# B&R Automation Studio project 8238 (part 30)

#### SupertrackLiftingStaticBag.st
```iecst
(* TODO: Add your comment here *)
FUNCTION_BLOCK SupertrackLiftingStaticBag

	messages ACCESS p_messages;

	// Device State Machine
	IF reset THEN
		IF rail_mt THEN
			udp_data.state := state := ReadyToReceive;
		ELSE
			udp_data.state := state := Loaded;
		END_IF;
	END_IF;
	IF udp_data.state = 0 THEN udp_data.state := state := ReadyToReceive; END_IF;

	// Debounce ON
	DBNC_up_timer(IN := up_raw, PT := DBNC_up_time);
	up := DBNC_up_timer.Q;

	DBNC_down_timer(IN := down_raw, PT := DBNC_down_time);
	down := DBNC_down_timer.Q;

	CASE udp_data.state OF
		Closed:
			IF dischargerRailSlingReady AND input_enabled AND NOT(safety_zone) AND NOT(halted) THEN
				udp_data.state := state := PreparingToLift;
			END_IF;

		PreparingToLift:
			IF PreparingToLiftTimer.Q THEN udp_data.state := state := Lifting; END_IF;

		Lifting:
			IF up THEN udp_data.state := state := DoneLifting; END_IF;

		DoneLifting:
			IF DoneLiftingTimer.Q THEN udp_data.state := state := InReceivePosition; END_IF;

		InReceivePosition:
			IF input_enabled AND NOT(safety_zone) AND NOT(halted) THEN
				udp_data.state := state := ReadyToReceive;
			ELSIF NOT(input_enabled) THEN
				udp_data.state := state := PreparingToLower;
			END_IF;

		ReadyToReceive:
			IF man_send THEN
				udp_data.state := state := Receiving;
			ELSIF NOT(input_enabled) OR safety_zone OR halted THEN
				udp_data.state := state := InReceivePosition;
			END_IF;

		Receiving:
			IF ReceivingTimer.Q THEN udp_data.state := state := PreparingToLower; END_IF;

		PreparingToLower:
			IF PreparingToLowerTimer.Q THEN udp_data.state := state := Lowering; END_IF;

		Lowering:
			IF down THEN udp_data.state := state := DoneLowering; END_IF;

		DoneLowering:
			IF DoneLoweringTimer.Q THEN
				IF rail_mt THEN
					udp_data.state := state := Closed;
				ELSE
					udp_data.state := state := Loaded;
				END_IF;
			END_IF;

		Loaded:
			IF NOT(halted) AND NOT(safety_zone) AND NOT(stopped) THEN
				udp_data.state := state := ReadyToTransfer;
			END_IF;

		ReadyToTransfer:
			IF open_signal OR man_open OR open_pendant THEN
				delete_latch := TRUE;
				udp_data.state := state := Unclamping;
			ELSIF halted OR stopped OR safety_zone THEN
				udp_data.state := state := Loaded;
			END_IF;

		Unclamping:
			IF UnclampingTimer.Q THEN udp_data.state := state := Opening; END_IF;

		Opening:
			IF static_open THEN udp_data.state := state := Transferring; END_IF;

		Transferring:
			IF man_send THEN udp_data.state := state := Closing; END_IF;

		Closing:
			IF static_close THEN udp_data.state := state := Closed; END_IF;

	END_CASE;

	clamp := udp_data.state = Unclamping OR udp_data.state = Opening OR udp_data.state = Transferring OR udp_data.state = Closing;
	open := udp_data.state = Opening;
	close := udp_data.state = Closing;

	lift_clamp := (
	udp_data.state = PreparingToLift
	OR udp_data.state = Lifting
	OR udp_data.state = PreparingToLower
	OR udp_data.state = Lowering
	);

	fire_up := (
	udp_data.state = Lifting
	OR udp_data.state = InReceivePosition
	OR udp_data.state = ReadyToReceive
	OR udp_data.state = Receiving
	OR udp_data.state = PreparingToLower
	);

	fire_down := NOT(fire_up);

	// Control Timers
	ReceivingTimer(IN := (udp_data.state = Receiving), PT := ReceivingTime);
	PreparingToLiftTimer(IN := (udp_data.state = PreparingToLift), PT := PreparingToLiftTime);
	PreparingToLowerTimer(IN := (udp_data.state = PreparingToLower), PT := PreparingToLowerTime);
	UnclampingTimer(IN := (udp_data.state = Unclamping), PT := UnclampingTime);
	DoneLiftingTimer(IN := udp_data.state = DoneLifting, PT := DoneLiftingTime);
	DoneLoweringTimer(IN := udp_data.state = DoneLowering, PT := DoneLoweringTime);

	// Comm Logic
	bring_ok := udp_data.state = Closing OR udp_data.state = Closed;
	waiting := FALSE;
	man_open := man_send := FALSE;
	sling_ready := udp_data.state = ReadyToTransfer;
	dischargerRailReceiveSignal := udp_data.state = DoneLowering;

	IF rail_mt THEN delete_latch := FALSE; END_IF;

	udp_data.alarm := alarm := FALSE;
	udp_data.warning_com.0 := warning_com.0 := FALSE;
	udp_data.warning_com.1 := warning_com.1 := FALSE;
	udp_data.warning_com.12 := warning_com.12 := delete_latch;
	udp_data.warning_com.14 := warning_com.14 := sling_ready;

	//messages.Write := 0;
	//IF UnexpectedBagTimer.Q   THEN messages.Write := BIT_SET(messages.Write,UNEXPECTED_BAG); END_IF;
	//IF MissingBagTimer.Q      THEN messages.Write := BIT_SET(messages.Write,MISSING_BAG); END_IF;

	// Always clear acknowledgements
	//brsmemset(ADR(messages.Read[0]),0,SIZEOF(messages.Read));

END_FUNCTION_BLOCK
```

#### SupertrackBinTransfer.st
```iecst
(* TODO: Add your comment here *)
FUNCTION_BLOCK SupertrackBinTransfer

	messages ACCESS p_messages;

	// Debounce Inputs
	DBNC_front_timer(IN := front_raw, PT := DBNC_front_time);
	front := DBNC_front_timer.Q;

	DBNC_arrive_timer(IN := arrive_raw, PT := DBNC_arrive_time);
	arrive := DBNC_arrive_timer.Q;

	DBNC_after_timer(IN := after_raw, PT := DBNC_after_time);
	after := DBNC_after_timer.Q;

	DBNC_mid_timer(IN := mid_raw, PT := DBNC_mid_time);
	mid_sensor := DBNC_mid_timer.Q;

	// Device State Machine
	IF reset THEN
		IF rail_mt AND NOT(going_to) THEN
			udp_data.state := state := ReadyToReceive;
		ELSIF NOT(rail_mt) THEN
			udp_data.state := state := ReadyToLoad;
		END_IF;
	END_IF;
	IF udp_data.state = 0 THEN udp_data.state := state := ReadyToReceive; END_IF;

	CASE udp_data.state OF
		ReadyToReceive:
			IF going_to THEN
				udp_data.state := state := Receiving;
			ELSIF NOT(rail_mt) THEN
				udp_data.state := state := ReadyToLoad;
			END_IF;

		Receiving:
			IF mid_sensor THEN
				udp_data.state := state := CatchRear;
			ELSIF NOT(going_to) THEN
				udp_data.state := state := ReadyToReceive;
			END_IF;

		CatchRear:
			IF NOT(rail_mt) THEN
				udp_data.state := state := ReadyToLoad;
			ELSIF NOT(going_to) THEN
				udp_data.state := state := ReadyToReceive;
			END_IF;

		ReadyToLoad:
			IF onoff AND NOT(halted) THEN
				udp_data.state := state := Stabilizing;
			ELSIF rail_mt AND NOT(front) THEN
				udp_data.state := state := ReadyToReceive;
			END_IF;

		Stabilizing:
			IF StabilizingTimer.Q THEN
				udp_data.state := state := BagReady;
			END_IF;

		BagReady:
			IF xfer_in_progress THEN
				udp_data.state := state := Loading;
			ELSIF man_send THEN
				udp_data.state := state := DeStabilizing;
			ELSIF rail_mt THEN
				udp_data.state := state := ReadyToReceive;
			END_IF;

		Loading:
			IF xfer_complete THEN
				udp_data.state := state := DeStabilizing;
			END_IF;

		DeStabilizing:
			IF DeStabilizingTimer.Q THEN
				udp_data.state := state := ReadyToRelease;
			END_IF;

		ReadyToRelease:
			IF fire_os THEN
				udp_data.state := state := ReleasingRear;
			END_IF;

		ReleasingRear:
			IF ReleaseRearTimer.Q THEN
				udp_data.state := state := Releasing;
			END_IF;

		Releasing:
			IF after OR NOT(fire) THEN
				udp_data.state := state := ReadyToReceive;
				man_send := FALSE;
			END_IF;

	END_CASE;

	// Comm Logic
	udp_data.waiting := waiting := (
	udp_data.state = ReadyToRelease
	AND front
	AND NOT(custom_send_lock)
	AND NOT(after)
	AND NOT(safety_zone)
	);

	udp_data.bring_ok := bring_ok := (
	udp_data.state = ReadyToReceive
	AND NOT(mid_sensor)
	AND NOT(arrive)
	AND NOT(going_to)
	AND NOT(custom_bring_lock)
	);

	IF going_to AND arrive THEN insert := TRUE; END_IF;

	// Control Timers
	StabilizingTimer(IN := (udp_data.state = Stabilizing), PT := StabilizingTime);
	DeStabilizingTimer(IN := (udp_data.state = DeStabilizing), PT := DeStabilizingTime);
	ReleaseRearTimer(IN := udp_data.state = ReleasingRear, PT := ReleaseRearTime);

	// Output Control
	front_stp := udp_data.state = Releasing;
	rear_stp := udp_data.state = Receiving OR udp_data.state = ReleasingRear OR udp_data.state = Releasing;
	stb := udp_data.state = Stabilizing OR udp_data.state = BagReady OR udp_data.state = Loading;
	fire_up := udp_data.state = Stabilizing OR udp_data.state = BagReady OR udp_data.state = Loading;

	sling_ready := udp_data.state = BagReady;

	// Alarm Timers
	AlarmTimer(IN := fire, PT := (t#1s * rail_alarm_time));
	UnexpectedBagTimer(IN := (front AND rail_mt), PT := UnexpectedBagTime);
	MissingBagTimer(IN := (NOT(front) AND NOT(rail_mt)), PT := MissingBagTime);

	// Alarm Coms
	udp_data.alarm := alarm := AlarmTimer.Q;
	udp_data.warning_com.0 := warning_com.0 := UnexpectedBagTimer.Q;
	udp_data.warning_com.1 := warning_com.1 := MissingBagTimer.Q;
	udp_data.warning_com.11 := warning_com.11 := udp_data.state = Loading;
	udp_data.warning_com.14 := warning_com.14 := sling_ready;

	//Rail Messages
	messages.Write := 0;
	//BAG_STUCK # not yet implemented
	IF UnexpectedBagTimer.Q THEN messages.Write := BIT_SET(messages.Write,UNEXPECTED_BAG); END_IF;
	IF MissingBagTimer.Q THEN messages.Write := BIT_SET(messages.Write,MISSING_BAG); END_IF;

	// Always clear acknowledgements
	brsmemset(ADR(messages.Read[0]),0,SIZEOF(messages.Read));

END_FUNCTION_BLOCK
```

#### SupertrackBinTransferWithNetComm.st
```iecst
(* TODO: Add your comment here *)
FUNCTION_BLOCK SupertrackBinTransferWithNetComm

	messages ACCESS p_messages;

	// Debounce Inputs
	DBNC_front_timer(IN := front_raw, PT := DBNC_front_time);
	front := DBNC_front_timer.Q;

	DBNC_arrive_timer(IN := arrive_raw, PT := DBNC_arrive_time);
	arrive := DBNC_arrive_timer.Q;

	DBNC_after_timer(IN := after_raw, PT := DBNC_after_time);
	after := DBNC_after_timer.Q;

	DBNC_mid_timer(IN := mid_raw, PT := DBNC_mid_time);
	mid_sensor := DBNC_mid_timer.Q;

	// Device State Machine
	IF reset THEN
		IF rail_mt AND NOT(going_to) THEN
			udp_data.state := state := ReadyToReceive;
		ELSIF NOT(rail_mt) THEN
			udp_data.state := state := ReadyToLoad;
		END_IF;
	END_IF;
	IF udp_data.state = 0 THEN udp_data.state := state := ReadyToReceive; END_IF;

	CASE udp_data.state OF
		ReadyToReceive:
			IF going_to THEN
				udp_data.state := state := Receiving;
			ELSIF NOT(rail_mt) THEN
				udp_data.state := state := ReadyToLoad;
			END_IF;

		Receiving:
			IF mid_sensor THEN
				udp_data.state := state := CatchRear;
			ELSIF NOT(going_to) THEN
				udp_data.state := state := ReadyToReceive;
			END_IF;

		CatchRear:
			IF NOT(rail_mt) THEN
				udp_data.state := state := ReadyToLoad;
			ELSIF NOT(going_to) THEN
				udp_data.state := state := ReadyToReceive;
			END_IF;

		ReadyToLoad:
			IF onoff AND NOT(halted) THEN
				udp_data.state := state := Stabilizing;
			ELSIF rail_mt AND NOT(front) THEN
				udp_data.state := state := ReadyToReceive;
			END_IF;

		Stabilizing:
			IF StabilizingTimer.Q THEN
				udp_data.state := state := BagReady;
			END_IF;

		BagReady:
			IF xfer_in_progress THEN
				udp_data.state := state := Loading;
			ELSIF man_send THEN
				udp_data.state := state := DeStabilizing;
			ELSIF rail_mt THEN
				udp_data.state := state := ReadyToReceive;
			END_IF;

		Loading:
			IF xfer_complete THEN
				udp_data.state := state := DeStabilizing;
			END_IF;

		DeStabilizing:
			IF DeStabilizingTimer.Q THEN
				udp_data.state := state := ReadyToRelease;
			END_IF;

		ReadyToRelease:
			IF fire_os THEN
				udp_data.state := state := ReleasingRear;
			END_IF;

		ReleasingRear:
			IF ReleaseRearTimer.Q THEN
				udp_data.state := state := Releasing;
			END_IF;

		Releasing:
			IF after OR NOT(fire) THEN
				udp_data.state := state := ReadyToReceive;
				man_send := FALSE;
			END_IF;

	END_CASE;

	// Comm Logic
	udp_data.waiting := waiting := (
	udp_data.state = ReadyToRelease
	AND front
	AND NOT(custom_send_lock)
	AND NOT(after)
	AND NOT(safety_zone)
	);

	udp_data.bring_ok := bring_ok := (
	udp_data.state = ReadyToReceive
	AND NOT(mid_sensor)
	AND NOT(arrive)
	AND NOT(going_to)
	AND NOT(custom_bring_lock)
	);

	IF going_to AND arrive THEN insert := TRUE; END_IF;

	// Control Timers
	StabilizingTimer(IN := (udp_data.state = Stabilizing), PT := StabilizingTime);
	DeStabilizingTimer(IN := (udp_data.state = DeStabilizing), PT := DeStabilizingTime);
	ReleaseRearTimer(IN := udp_data.state = ReleasingRear, PT := ReleaseRearTime);

	// Output Control
	front_stp := udp_data.state = Releasing;
	rear_stp := udp_data.state = Receiving OR udp_data.state = ReleasingRear OR udp_data.state = Releasing;
	stb := udp_data.state = Stabilizing OR udp_data.state = BagReady OR udp_data.state = Loading;
	fire_up := udp_data.state = Stabilizing OR udp_data.state = BagReady OR udp_data.state = Loading;

	sling_ready := udp_data.state = BagReady;

	// Alarm Timers
	AlarmTimer(IN := fire, PT := (t#1s * rail_alarm_time));
	UnexpectedBagTimer(IN := (front AND rail_mt), PT := UnexpectedBagTime);
	MissingBagTimer(IN := (NOT(front) AND NOT(rail_mt)), PT := MissingBagTime);

	// Alarm Coms
	udp_data.alarm := alarm := AlarmTimer.Q;
	udp_data.warning_com.0 := warning_com.0 := UnexpectedBagTimer.Q;
	udp_data.warning_com.1 := warning_com.1 := MissingBagTimer.Q;

	//Rail Messages
	messages.Write := 0;
	//BAG_STUCK # not yet implemented
	IF UnexpectedBagTimer.Q THEN messages.Write := BIT_SET(messages.Write,UNEXPECTED_BAG); END_IF;
	IF MissingBagTimer.Q THEN messages.Write := BIT_SET(messages.Write,MISSING_BAG); END_IF;

	// Always clear acknowledgements
	brsmemset(ADR(messages.Read[0]),0,SIZEOF(messages.Read));

END_FUNCTION_BLOCK
```

#### SupertrackBeltConveyor.st
```iecst
(* TODO: Add your comment here *)
FUNCTION_BLOCK SupertrackBeltConveyor

	messages ACCESS p_messages;

	// Debounce Inputs
	DBNC_front_timer(IN := front_raw, PT := DBNC_front_time);
	front := DBNC_front_timer.Q;

	DBNC_arrive_timer(IN := arrive_raw, PT := DBNC_arrive_time);
	arrive := DBNC_arrive_timer.Q;

	DBNC_after_timer(IN := after_raw, PT := DBNC_after_time);
	after := DBNC_after_timer.Q;

	// Device State Machine
	IF reset THEN udp_data.state := state := ReadyToWork; END_IF;
	IF udp_data.state = 0 THEN udp_data.state := state := ReadyToWork; END_IF;

	CASE udp_data.state OF
		ReadyToWork:
			IF NOT(rail_mt) AND NOT(halted) THEN
				udp_data.state := state := RunToFront;
			END_IF;

		RunToFront:
			IF NOT(front) THEN
				udp_data.state := state := ReadyToRelease;
			END_IF;

		ReadyToRelease:
			IF fire_os THEN
				udp_data.state := state := Releasing;
			END_IF;

		Releasing:
			IF after OR NOT(fire) THEN
				udp_data.state := state := ClearBelt;
			END_IF;

		ClearBelt:
			IF ClearBeltTimer.Q THEN
				udp_data.state := state := ReadyToWork;
			END_IF;

	END_CASE;

	// Comm Logic
	udp_data.waiting := waiting := (
	udp_data.state = ReadyToRelease
	AND NOT(custom_send_lock)
	AND NOT(safety_zone)
	);

	udp_data.bring_ok := bring_ok := (
	udp_data.state = ReadyToWork
	AND arrive
	AND front
	AND NOT(going_to)
	AND NOT(custom_bring_lock)
	);

	IF going_to AND NOT(arrive) THEN insert := TRUE; END_IF;

	// Output Control
	run_conveyor := (
	NOT(halted) AND NOT halt
	AND (
	udp_data.state = Releasing
	OR udp_data.state = ClearBelt
	OR udp_data.state = RunToFront
	OR (going_to AND front AND (udp_data.state = ReadyToWork))
	));

	releasing := (
	udp_data.state = Releasing
	OR udp_data.state = ClearBelt
	);

	//Control Timers
	ClearBeltTimer(IN := (udp_data.state = ClearBelt AND arrive AND NOT receiving AND conveyor_running AND front AND NOT(fire)), PT := ClearBeltTime);
	MaximumBeltRunningTime(IN:= (run_conveyor AND conveyor_running), PT := MaximumRunningTime );
	IF MaximumBeltRunningTime.Q THEN
		halt := TRUE;
	END_IF;

	// Alarm Timers
	AlarmTimer(IN := fire, PT := (t#1s * rail_alarm_time));
	UnexpectedBagTimer(IN := (NOT front AND ((rail_mt AND (udp_data.state <> ClearBelt)) OR (conveyor_running AND (udp_data.state = ClearBelt)))) , PT := UnexpectedBagTime);
	MissingBagTimer(IN := (front AND NOT(rail_mt)), PT := MissingBagTime );

	// Alarm Coms
	udp_data.alarm := alarm := AlarmTimer.Q;
	udp_data.warning_com.0 := warning_com.0 := 0;//UnexpectedBagTimer.Q;
	udp_data.warning_com.1 := warning_com.1 := 0;//MissingBagTimer.Q;

	//Rail Messages
	messages.Write := 0;
	//BAG_STUCK # not yet implemented
	IF UnexpectedBagTimer.Q THEN messages.Write := BIT_SET(messages.Write,UNEXPECTED_BAG); END_IF;
	IF MissingBagTimer.Q THEN messages.Write := BIT_SET(messages.Write,MISSING_BAG); END_IF;
	IF halt THEN  messages.Write := BIT_SET(messages.Write,EXCEED_RUN_TIME); END_IF;

	CASE messages.Read[EXCEED_RUN_TIME] OF
		1: //They want to continue running
			halt := 0;
		2: //Confirm belt is clear
			halt := 0;
			IF (udp_data.state = RunToFront) THEN
				IF rail_mt THEN
					udp_data.state := state := ReadyToWork;
				END_IF;
			ELSE
				udp_data.state := state := ReadyToWork;
			END_IF;
	END_CASE;

	// Always clear acknowledgements
	brsmemset(ADR(messages.Read[0]),0,SIZEOF(messages.Read));

END_FUNCTION_BLOCK
```

#### SupertrackPrimaryLoadingPoint.st
```iecst
(* TODO: Add your comment here *)
FUNCTION_BLOCK SupertrackPrimaryLoadingPoint

	messages ACCESS p_messages;
	loadcell ACCESS p_loadcell;

	// Debounce Inputs
	DBNC_front_timer(IN := front_raw, PT := DBNC_front_time);
	front := DBNC_front_timer.Q;

	// Device State Machine
	IF reset THEN
		IF front THEN
			udp_data.state := state := Loading;
		ELSE
			udp_data.state := state := ReadyToWork;
		END_IF;
	END_IF;
	IF udp_data.state = 0 THEN udp_data.state := state := ReadyToWork; END_IF;

	CASE udp_data.state OF
		ReadyToWork:
			IF front AND onoff AND NOT(halted) THEN
				udp_data.state := state := Loading;
			END_IF;

		Loading:
			IF man_send OR EDGENEG(foot) THEN
				man_send := 0;
				udp_data.state := state := ReadyToRelease;
			ELSIF rail_mt AND NOT front_raw THEN
				udp_data.state := state := ReadyToWork;
			END_IF;

		ReadyToRelease:
			IF fire_os THEN
				udp_data.state := state := Releasing;
			END_IF;

		Releasing:
			IF NOT(fire) THEN
				udp_data.state := state := ReadyToWork;
			END_IF;

	END_CASE;

	// Comm Logic
	udp_data.waiting := waiting := (
	udp_data.state = ReadyToRelease
	AND NOT(custom_send_lock)
	AND NOT(safety_zone)
	AND NOT(loadcell.over_weight)
	);

	udp_data.bring_ok := bring_ok := (
	udp_data.state = ReadyToWork
	AND NOT(arrive)
	AND NOT(custom_bring_lock)
	);

	IF going_to AND arrive THEN insert := TRUE; END_IF;

	// Input Control
	arrive := arrive_raw := front_raw;

	// Weight
	IF NOT(udp_data.state = Releasing) THEN
		loadcell.capture_weight_bool := TRUE;
	ELSE
		loadcell.capture_weight_bool := FALSE;
	END_IF;

	// Output Control
	stp := (udp_data.state = Releasing);  // Stop inside remover

	// Alarm Timers
	AlarmTimer(IN := fire, PT := (t#1s * rail_alarm_time));
	UnexpectedBagTimer(IN := (front AND rail_mt), PT := UnexpectedBagTime);

	// Alarm Coms
	alarm := AlarmTimer.Q;
	warning_com.0 := UnexpectedBagTimer.Q;

	//Rail Messages
	messages.Write := 0;
	//BAG_STUCK # not yet implemented
	IF UnexpectedBagTimer.Q THEN messages.Write := BIT_SET(messages.Write,UNEXPECTED_BAG); END_IF;

	// Always clear acknowledgements
	brsmemset(ADR(messages.Read[0]),0,SIZEOF(messages.Read));

END_FUNCTION_BLOCK
```

#### SupertrackBagCloserTracked.st
```iecst
(* TODO: Add your comment here *)
FUNCTION_BLOCK SupertrackBagCloserTracked

	messages ACCESS p_messages;

	// Debounce Inputs
	DBNC_front_timer(IN := front_raw, PT := DBNC_front_time);
	front := DBNC_front_timer.Q;

	DBNC_arrive_timer(IN := arrive_raw, PT := DBNC_arrive_time);
	arrive := DBNC_arrive_timer.Q;

	DBNC_after_timer(IN := after_raw, PT := DBNC_after_time);
	after := DBNC_after_timer.Q;

	// Device State Machine
	IF reset THEN udp_data.state := state := ReadyToWork; END_IF;
	IF udp_data.state = 0 THEN udp_data.state := state := ReadyToWork; END_IF;

	CASE udp_data.state OF
		ReadyToWork:
			IF NOT(rail_mt) AND front AND onoff AND NOT(halted) THEN
				udp_data.state := state := Stabilizing;
			END_IF;

		Stabilizing:
			IF StabilizingTimer.Q THEN
				udp_data.state := state := Opening;
			ELSIF NOT(onoff) THEN
				udp_data.state := state := ReadyToWork;
			END_IF;

		Opening:
			IF OpeningTimer.Q THEN
				udp_data.state := state := Closing;
			END_IF;

		Closing:
			IF ClosingTimer.Q THEN
				udp_data.state := state := Destabilizing;
			END_IF;

		Destabilizing:
			IF DestabilizingTimer.Q THEN
				IF empty_bag THEN
					udp_data.state := state := ReadyToRelease;
				ELSIF (messages.Read[BAG_NOT_CLOSED] = 2) THEN
					udp_data.state := state := ReadyToRelease;
				ELSIF (messages.Read[BAG_NOT_CLOSED] = 1) THEN
					udp_data.state := state := Stabilizing;
				END_IF;
			END_IF;

		ReadyToRelease:
			IF fire_os THEN
				udp_data.state := state := Releasing;
			END_IF;

		Releasing:
			IF after OR NOT(fire) THEN
				udp_data.state := state := ReadyToWork;
			END_IF;

	END_CASE;

	// Comm Logic
	udp_data.waiting := waiting := (
	udp_data.state = ReadyToRelease
	AND NOT(custom_send_lock)
	AND NOT(after)
	AND NOT(safety_zone)
	);

	udp_data.bring_ok := bring_ok := (
	udp_data.state = ReadyToWork
	AND NOT(arrive)
	AND NOT(going_to)
	AND NOT(custom_bring_lock)
	);

	IF going_to AND arrive THEN insert := TRUE; END_IF;

	// Output Control
	stb := (
	udp_data.state = Stabilizing
	OR udp_data.state = Opening
	OR udp_data.state = Closing
	);

	open := (
	udp_data.state = Opening
	OR udp_data.state = Closing
	);

	stp := udp_data.state = Releasing;
	close := udp_data.state = Closing;

	// Control Timers

	StabilizingTimer(IN := (udp_data.state = Stabilizing), PT := StabilizingTime);
	DestabilizingTimer(IN := (udp_data.state = Destabilizing), PT := DestabilizingTime);
	ClosingTimer(IN := (udp_data.state = Closing), PT := ClosingTime);
	OpeningTimer(IN := (udp_data.state = Opening), PT := OpeningTime);

	// Alarm Timers
	AlarmTimer(IN := fire, PT := (t#1s * rail_alarm_time));
	UnexpectedBagTimer(IN := (front AND rail_mt), PT := UnexpectedBagTime);
	MissingBagTimer(IN := (NOT(front) AND NOT(rail_mt)), PT := MissingBagTime);
	BagNotClosedTimer(IN := ((udp_data.state = Destabilizing) AND NOT empty_bag), PT := BagNotClosedTime);

	udp_data.alarm := alarm := AlarmTimer.Q;
	udp_data.warning_com.0 := warning_com.0 := 0;//UnexpectedBagTimer.Q;
	udp_data.warning_com.1 := warning_com.1 := 0;//MissingBagTimer.Q;

	// Rail Fault Handling.
	messages.Write := 0;
	//BAG_STUCK  -- NOT YET IMPLEMENTED
	IF UnexpectedBagTimer.Q   THEN messages.Write := BIT_SET(messages.Write,UNEXPECTED_BAG); END_IF;
	IF MissingBagTimer.Q      THEN messages.Write := BIT_SET(messages.Write,MISSING_BAG); END_IF;
	IF BagNotClosedTimer.Q    THEN messages.Write := BIT_SET(messages.Write,BAG_NOT_CLOSED); END_IF;

	// Always clear acknowledgements
	brsmemset(ADR(messages.Read[0]),0,SIZEOF(messages.Read));

END_FUNCTION_BLOCK
```

#### SupertrackBagCloserUnTracked.st
```iecst
(* TODO: Add your comment here *)
FUNCTION_BLOCK SupertrackBagCloserUnTracked

	messages ACCESS p_messages;

	// Debounce Inputs
	DBNC_front_timer(IN := front_raw, PT := DBNC_front_time);
	front := DBNC_front_timer.Q;

	DBNC_arrive_timer(IN := arrive_raw, PT := DBNC_arrive_time);
	arrive := DBNC_arrive_timer.Q;

	DBNC_after_timer(IN := after_raw, PT := DBNC_after_time);
	after := DBNC_after_timer.Q;

	// Device State Machine
	IF reset THEN udp_data.state := state := ReadyToWork; END_IF;
	IF udp_data.state = 0 THEN udp_data.state := state := ReadyToWork; END_IF;

	CASE udp_data.state OF
		ReadyToWork:
			IF front AND onoff AND NOT(halted) THEN
				udp_data.state := state := Stabilizing;
			END_IF;

		Stabilizing:
			IF StabilizingTimer.Q THEN
				udp_data.state := state := Opening;
			ELSIF NOT(onoff) THEN
				udp_data.state := state := ReadyToWork;
			END_IF;

		Opening:
			IF OpeningTimer.Q THEN
				udp_data.state := state := Closing;
			END_IF;

		Closing:
			IF ClosingTimer.Q THEN
				udp_data.state := state := Destabilizing;
			END_IF;

		Destabilizing:
			IF DestabilizingTimer.Q THEN
				IF empty_bag THEN
					udp_data.state := state := ReadyToRelease;
				ELSIF (messages.Read[BAG_NOT_CLOSED] = 2) THEN
					udp_data.state := state := ReadyToRelease;
				ELSIF (messages.Read[BAG_NOT_CLOSED] = 1) THEN
					udp_data.state := state := Stabilizing;
				END_IF;
			END_IF;

		ReadyToRelease:
			IF fire_os THEN
				udp_data.state := state := Releasing;
			END_IF;

		Releasing:
			IF after OR NOT(fire) THEN
				udp_data.state := state := ReadyToWork;
			END_IF;

	END_CASE;

	// Comm Logic
	udp_data.waiting := waiting := (
	udp_data.state = ReadyToRelease
	AND NOT(custom_send_lock)
	AND NOT(after)
	AND NOT(safety_zone)
	);

	udp_data.bring_ok := bring_ok := (
	udp_data.state = ReadyToWork
	AND NOT(arrive)
	AND NOT(going_to)
	AND NOT(custom_bring_lock)
	);

	IF going_to AND arrive THEN insert := TRUE; END_IF;

	// Output Control
	stb := (
	udp_data.state = Stabilizing
	OR udp_data.state = Opening
	OR udp_data.state = Closing
	);

	open := (
	udp_data.state = Opening
	OR udp_data.state = Closing
	);

	stp := udp_data.state = Releasing;
	close := udp_data.state = Closing;

	// Control Timers

	StabilizingTimer(IN := (udp_data.state = Stabilizing), PT := StabilizingTime);
	DestabilizingTimer(IN := (udp_data.state = Destabilizing), PT := DestabilizingTime);
	ClosingTimer(IN := (udp_data.state = Closing), PT := ClosingTime);
	OpeningTimer(IN := (udp_data.state = Opening), PT := OpeningTime);

	// Alarm Timers
	AlarmTimer(IN := fire, PT := (t#1s * rail_alarm_time));
	udp_data.alarm := alarm := AlarmTimer.Q;

	// Rail Fault Handling.
	messages.Write := 0;
	//BAG_STUCK  -- NOT YET IMPLEMENTED
	IF UnexpectedBagTimer.Q   THEN messages.Write := BIT_SET(messages.Write,UNEXPECTED_BAG); END_IF;
	IF MissingBagTimer.Q      THEN messages.Write := BIT_SET(messages.Write,MISSING_BAG); END_IF;
	IF BagNotClosedTimer.Q    THEN messages.Write := BIT_SET(messages.Write,BAG_NOT_CLOSED); END_IF;

	// Always clear acknowledgements
	brsmemset(ADR(messages.Read[0]),0,SIZEOF(messages.Read));

END_FUNCTION_BLOCK
```

#### SupertrackSplitRailTransfer.st
```iecst
(* TODO: Add your comment here *)
FUNCTION_BLOCK SupertrackSplitRailTransfer

	messages ACCESS p_messages;

	// Debounce Inputs
	DBNC_front_timer(IN := front_raw, PT := DBNC_front_time);
	front := DBNC_front_timer.Q;

	DBNC_arrive_timer(IN := arrive_raw, PT := DBNC_arrive_time);
	arrive := DBNC_arrive_timer.Q;

	DBNC_after_timer(IN := after_raw, PT := DBNC_after_time);
	after := DBNC_after_timer.Q;

	DBNC_before_timer(IN := before_raw, PT := DBNC_before_time);
	before := DBNC_before_timer.Q;

	// Device State Machine
	IF reset THEN
		udp_data.state := state := ReadyToWork;
		man_send := FALSE;
	END_IF;
	IF udp_data.state = 0 THEN udp_data.state := state := ReadyToWork; END_IF;

	CASE udp_data.state OF
		ReadyToWork:
			IF NOT(rail_mt) AND front AND onoff AND NOT(halted) THEN
				udp_data.state := state := Stabilizing;
			END_IF;

		Stabilizing:
			IF StabilizingTimer.Q THEN
				udp_data.state := state := ReadyForTransfer;
			END_IF;

		ReadyForTransfer:
			IF xfer_complete OR man_send OR open_signal THEN
				udp_data.state := state := Destabilizing;
			END_IF;

		Destabilizing:
			IF DestabilizingTimer.Q THEN
				IF over_full_sensor THEN
					udp_data.state := state := Overfull;
				ELSE
					udp_data.state := state := ReadyToRelease;
				END_IF;
			END_IF;

		Overfull:
			IF NOT(over_full_sensor) THEN
				udp_data.state := state := ReadyToRelease;
			END_IF;

		ReadyToRelease:
			IF fire_os THEN
				man_send := FALSE;
				udp_data.state := state := Releasing;
			END_IF;

		Releasing:
			IF NOT(fire) THEN
				udp_data.state := state := ReadyToWork;
			ELSIF after_b OR after_a THEN
				udp_data.state := state := ReleaseRear;
			END_IF;

		ReleaseRear:
			IF NOT(fire) OR after THEN
				udp_data.state := state := ReadyToWork;
			END_IF;

	END_CASE;

	// Comm Logic
	udp_data.waiting := waiting := (
	udp_data.state = ReadyToRelease
	AND front
	AND NOT(custom_send_lock)
	AND NOT(before)
	AND NOT(after)
	AND NOT(over_full_sensor)
	AND NOT(safety_zone)
	);

	udp_data.bring_ok := bring_ok := (
	udp_data.state = ReadyToWork
	AND NOT(before)
	AND NOT(arrive)
	AND NOT(going_to)
	AND NOT(custom_bring_lock)
	AND NOT(stp)
	);

	//Insert
	IF going_to AND arrive THEN insert := TRUE; END_IF;

	// Input Control
	arrive_raw := front_raw := front_a AND front_b;

	// Output Control
	stb := udp_data.state = Stabilizing OR udp_data.state = ReadyForTransfer;
	foot := FootDelayTimer.Q;
	stp := udp_data.state = Releasing;
	sling_ready := transfer_requested_signal AND udp_data.state = ReadyForTransfer AND onoff AND NOT(halted) AND NOT(safety_zone);
	over_full_light := over_full_sensor;
	stp_a := udp_data.state = ReleaseRear;

	// Output Switch Control
	IF SwInARTrig.Q THEN
		sw_in_a := TRUE;
	END_IF;

	IF before AND going_to THEN
		sw_in_a := FALSE;
		sw_in_b  := TRUE;
	END_IF;

	IF NOT(going_to) THEN
		sw_in_a := FALSE;
		sw_in_b  := FALSE;
	END_IF;

	IF SwOutARTrig.Q THEN
		sw_out_a := TRUE;
	END_IF;

	IF fire AND after THEN
		sw_out_a := FALSE;
		sw_out_b  := TRUE;
	END_IF;

	IF NOT(fire) THEN
		sw_out_a := FALSE;
		sw_out_b  := FALSE;
	END_IF;

	IF reset THEN
		sw_out_a := FALSE;
		sw_out_b  := FALSE;
	END_IF;

	// Control Timers
	StabilizingTimer(IN := udp_data.state = Stabilizing, PT := StabilizingTime);
	FootDelayTimer(IN := stb, PT := FootDelayTime);
	DestabilizingTimer(IN := udp_data.state = Destabilizing, PT := DestabilizingTime);

	// Control Triggers
	SwInARTrig(CLK := (going_to));
	SwOutARTrig(CLK := (fire));

	// Alarm Timers
	AlarmTimer(IN := fire, PT := (t#1s * rail_alarm_time));
	UnexpectedBagTimer(IN := (front AND rail_mt), PT := UnexpectedBagTime);
	MissingBagTimer(IN := (NOT(front) AND NOT(rail_mt)), PT := MissingBagTime);

	udp_data.alarm := AlarmTimer.Q;
	udp_data.warning_com.0 := warning_com.0 := UnexpectedBagTimer.Q;
	udp_data.warning_com.1 := warning_com.1 := MissingBagTimer.Q;
	udp_data.warning_com.11 := warning_com.11 := xfer_in_progress;
	udp_data.warning_com.14 := warning_com.14 := sling_ready;

	//Rail Messages
	messages.Write := 0;
	//BAG_STUCK # not yet implemented
	IF UnexpectedBagTimer.Q THEN messages.Write := BIT_SET(messages.Write,UNEXPECTED_BAG); END_IF;
	IF MissingBagTimer.Q THEN messages.Write := BIT_SET(messages.Write,MISSING_BAG); END_IF;

	// Always clear acknowledgements
	brsmemset(ADR(messages.Read[0]),0,SIZEOF(messages.Read));

END_FUNCTION_BLOCK
```

#### SupertrackRatchetLift.st
```iecst
(* TODO: Add your comment here *)
FUNCTION_BLOCK SupertrackRatchetLift

	messages ACCESS p_messages;

	// Debounce Inputs
	DBNC_arrive_timer(IN := arrive_raw, PT := DBNC_arrive_time);
	arrive := DBNC_arrive_timer.Q;

	DBNC_after_timer(IN := after_raw, PT := DBNC_after_time);
	after := DBNC_after_timer.Q;

	// Device State Machine
	IF reset THEN udp_data.state := state := ReadyToWork; END_IF;
	IF udp_data.state = 0 THEN udp_data.state := state := ReadyToWork; END_IF;

	CASE udp_data.state OF
		ReadyToWork:
			IF NOT(rail_mt) AND onoff AND NOT(halted) THEN
				udp_data.state := state := ReadyToRelease;
			END_IF;

		ReadyToRelease:
			IF fire_os THEN
				udp_data.state := state := Retract;
			END_IF;

		Retract:
			IF LowSensorTimer.Q THEN
				udp_data.state := state := Extend;
			END_IF;

		Extend:
			IF HighSensorTimer.Q THEN
				udp_data.state := state := Retract2;
			END_IF;

		Retract2:
			IF LowSensorTimer.Q THEN
				udp_data.state := state := Releasing;
			END_IF;

		Releasing:
			IF after OR NOT(fire) THEN
				udp_data.state := state := ReadyToWork;
			END_IF;
	END_CASE;

	// Comm Logic
	udp_data.waiting := waiting := (
	udp_data.state = ReadyToRelease
	AND rail_full
	AND NOT(custom_send_lock)
	AND NOT(after)
	AND NOT(safety_zone)
	);

	udp_data.bring_ok := bring_ok := (
	udp_data.state = ReadyToWork
	AND rail_mt
	AND high_valve
	AND NOT(arrive)
	AND NOT(going_to)
	AND NOT(custom_bring_lock)
	);

	IF going_to AND arrive THEN insert := TRUE; END_IF;

	// Output Control
	ratchet := udp_data.state = Retract OR udp_data.state = Retract2;

	//Output Timer
	HighSensorTimer(IN := high_valve, PT := HighSensorTime);
	LowSensorTimer(IN := low_valve, PT := LowSensorTime);

	// Alarm Timers
	AlarmTimer(IN := fire, PT := (t#1s * rail_alarm_time));
	UnexpectedBagTimer(IN := (arrive AND rail_mt AND NOT(ratchet)), PT := UnexpectedBagTime);

	// Alarm Coms
	udp_data.alarm := alarm := AlarmTimer.Q;
	udp_data.warning_com.0 := warning_com.0 := UnexpectedBagTimer.Q;

	messages.Write := 0;
	IF UnexpectedBagTimer.Q   THEN messages.Write := BIT_SET(messages.Write,UNEXPECTED_BAG); END_IF;

	// Always clear acknowledgements
	brsmemset(ADR(messages.Read[0]),0,SIZEOF(messages.Read));

END_FUNCTION_BLOCK
```

#### SupertrackRotasort.st
```iecst
(* TODO: Add your comment here *)
FUNCTION_BLOCK SupertrackRotasort

	messages ACCESS p_messages;
	loadcell ACCESS p_loadcell;

	// Debounce Inputs
	DBNC_before_timer(IN := before_raw, PT := DBNC_before_time);
	before := DBNC_before_timer.Q;

	DBNC_loading_position_timer(IN := loading_position_raw, PT := DBNC_loading_position_time);
	loading_position := DBNC_loading_position_timer.Q;

	DBNC_after_timer(IN := after_raw, PT := DBNC_after_time);
	after := DBNC_after_timer.Q;

	// Device State Machine
	IF reset THEN udp_data.state := state := Reset; END_IF;
	IF udp_data.state = 0 THEN udp_data.state := state := Reset; END_IF;

	CASE udp_data.state OF

		Reset: //decide what to do
			IF onoff AND NOT(halted) THEN
				IF going_to THEN
					udp_data.state := state := Receiving;
				ELSIF (loading_position_raw OR NOT rail_mt) THEN
					udp_data.state := state := Loading;
				ELSIF rail_mt AND NOT front_a AND NOT front_b AND NOT loading_position_raw THEN
					udp_data.state := state := ReadyToReceive;
				ELSIF ton_straight.Q THEN
					udp_data.state := state := ReadyToReceive;
				END_IF;
			END_IF;

		ReadyToReceive: // stp a & b are open waiting for bags to pass through.
			IF going_to THEN
				udp_data.state := state := Receiving;
			END_IF;

		Receiving: //Bag is on its way  stp b is open wait for bag to arrive.
			IF arrive THEN
				udp_data.state := state := SettleOnPoints;
			END_IF;

		SettleOnPoints:  //Wait for bag to arrive a and b closed
			IF ton_settledOnPoints.Q THEN
				udp_data.state := state := MoveToRotateBagIn;
			END_IF;

		MoveToRotateBagIn: // Move to "in" position
			IF ton_rotated.Q THEN
				udp_data.state := state := ReleaseBagToLoading;
			END_IF;

		ReleaseBagToLoading: // Release the bag in the loading position
			IF loading_position THEN
				udp_data.state := state := Loading;
			END_IF;

		Loading:
			IF loadcell.over_weight THEN
				udp_data.state := state := OverWeight;
			ELSIF NearWeightTimer.Q THEN
				udp_data.state := state := NearWeight;
			ELSIF man_send THEN
				udp_data.state := state := ReadyToRelease;
			END_IF;

		NearWeight:
			IF loadcell.over_weight THEN
				udp_data.state := state := OverWeight;
			ELSIF (FullWeightTimer.Q OR man_send) THEN
				udp_data.state := state := ReadyToRelease;
			END_IF;

		OverWeight:
			IF NOT(loadcell.over_weight) THEN
				udp_data.state := state := Loading;
			END_IF;

		ReadyToRelease:// Wait for the decider to tell us wehere to go
			IF fire_os THEN
				udp_data.state := state := MoveToRotateBagOut;
			END_IF;

		MoveToRotateBagOut: // Rotate so we can release a bag.
			IF ton_rotated.Q THEN
				udp_data.state := state := ReleaseBagToPoints;
			END_IF;

		ReleaseBagToPoints: //
			IF front_a AND front_b THEN
				udp_data.state := state := RetractPusher;
			END_IF;

		RetractPusher: //
			IF ton_retractPusher.Q THEN
				udp_data.state := state := MoveToStraightBagOut;
			END_IF;

		MoveToStraightBagOut:
			IF ton_straight.Q THEN
				udp_data.state := state := Releasing;
			END_IF;

		Releasing:
			IF after OR NOT(fire) THEN
				udp_data.state := state := Reset;
			END_IF;
	END_CASE;

	// Comm Logic
	udp_data.waiting := waiting := (
	udp_data.state = ReadyToRelease
	AND NOT(custom_send_lock)
	AND NOT(after)
	AND NOT(safety_zone)
	AND sort_exit_clear
	AND onoff
	);

	udp_data.bring_ok := bring_ok := (
	udp_data.state = ReadyToReceive
	AND ton_straight.Q
	AND NOT(front_a)
	AND NOT(front_b)
	AND NOT(going_to)
	AND NOT(custom_bring_lock)
	AND NOT(loading_position)
	AND sort_entry_clear
	AND onoff
	);

	//Don't arrive the bag until we are in the loading position and points are back straight.
	IF going_to AND (loading_position AND ton_straight.Q) THEN insert := TRUE; END_IF;

	// Input Control
	front := front_a OR front_b;
	arrive := arrive_raw;

	// Output Control
	stp_a := (
	((udp_data.state = ReadyToReceive) AND ton_straight.Q)
	OR ((udp_data.state = Loading) AND ton_straight.Q)
	OR ((udp_data.state = NearWeight) AND ton_straight.Q)
	OR ((udp_data.state = ReadyToRelease) AND ton_straight.Q)
	OR ((udp_data.state = ReleaseBagToLoading) AND ton_rotated.Q)
	OR ((udp_data.state = ReleaseBagToPoints) AND ton_rotated.Q)
	OR ((udp_data.state = Releasing) AND ton_straight.Q)
	OR ((udp_data.state = Reset) AND NOT onoff AND ton_straight.Q)
	);

	stp_b := (
	((udp_data.state = ReadyToReceive) AND ton_straight.Q)
	OR ((udp_data.state = Receiving) AND ton_straight.Q)
	OR ((udp_data.state = Loading) AND ton_straight.Q)
	OR ((udp_data.state = NearWeight) AND ton_straight.Q)
	OR ((udp_data.state = ReadyToRelease) AND ton_straight.Q)
	OR ((udp_data.state = ReleaseBagToLoading) AND ton_rotated.Q)
	OR ((udp_data.state = ReleaseBagToPoints) AND ton_rotated.Q)
	OR ((udp_data.state = Releasing) AND ton_straight.Q)
	OR ((udp_data.state = Reset) AND NOT onoff AND ton_straight.Q)
	);

	rotate := (
	(udp_data.state = MoveToRotateBagIn)
	OR (udp_data.state = ReleaseBagToLoading)
	OR (udp_data.state = MoveToRotateBagOut)
	OR (udp_data.state = ReleaseBagToPoints)
	OR (udp_data.state = RetractPusher)
	);

	switch := rotate;// AND NOT ton_rotated.Q;
	reset_switch  := NOT rotate;// AND NOT ton_straight.Q;
	foot := (udp_data.state = Loading);

	pusher := (udp_data.state = ReleaseBagToPoints); // Pusher pushes the bag out.
	clamp := ((rotate AND NOT ton_rotated.Q) OR (NOT rotate AND NOT ton_straight.Q));  // We have to fire this to unlock the rails so we can move them

	// Output Switch Control
	IF SwInARTrig.Q THEN
		sw_in_a := TRUE;
	END_IF;

	IF before AND going_to THEN
		sw_in_a := FALSE;
		sw_in_b  := TRUE;
	END_IF;

	IF NOT(going_to) THEN
		sw_in_a := FALSE;
		sw_in_b  := FALSE;
	END_IF;

	IF SwOutARTrig.Q THEN
		sw_out_a := TRUE;
	END_IF;

	IF fire AND after THEN
		sw_out_a := FALSE;
		sw_out_b  := TRUE;
	END_IF;

	IF NOT(fire) THEN
		sw_out_a := FALSE;
		sw_out_b  := FALSE;
	END_IF;

	IF reset THEN
		sw_out_a := FALSE;
		sw_out_b  := FALSE;
	END_IF;

	// Control Triggers
	SwInARTrig(CLK := (going_to));
	SwOutARTrig(CLK := (fire));

	ton_straight(IN:= sw_in_a AND sw_in_b, PT:= rotateTime);
	ton_rotated(IN:= sw_out_a AND sw_out_b, PT:= rotateTime);
	ton_settledOnPoints(IN:= front_a AND front_b, PT:= settleTime);
	ton_retractPusher(IN:=(udp_data.state = RetractPusher), PT:= retractTime);

	// Weight Comm
	IF (udp_data.state = NearWeight) OR (udp_data.state = ReadyToRelease) OR (udp_data.state = Loading) OR (udp_data.state = OverWeight)THEN
		loadcell.capture_weight_bool := TRUE;
	ELSE
		loadcell.capture_weight_bool := FALSE;
	END_IF;

	NearWeightTimer(IN := (loadcell.near_weight), PT := NearWeightTime);
	FullWeightTimer(IN := (loadcell.full), PT := FullWeightTime);

	// Input Control
	man_send := FALSE;
	IF man_send_button THEN
		man_send := TRUE;
	END_IF;

	// Alarm Timers
	AlarmTimer(IN := fire, PT := (t#1s * rail_alarm_time));
	UnexpectedBagTimer(IN := (loading_position AND rail_mt), PT := UnexpectedBagTime);
	MissingBagTimer(IN := (NOT(loading_position) AND NOT(rail_mt)), PT := MissingBagTime);

	// Alarm Coms
	alarm := AlarmTimer.Q;
	warning_com.0 := UnexpectedBagTimer.Q;
	warning_com.1 := MissingBagTimer.Q;

	//Rail Messages
	messages.Write := 0;
	//BAG_STUCK # not yet implemented
	IF UnexpectedBagTimer.Q THEN messages.Write := BIT_SET(messages.Write,UNEXPECTED_BAG); END_IF;
	IF MissingBagTimer.Q THEN messages.Write := BIT_SET(messages.Write,MISSING_BAG); END_IF;

	// Always clear acknowledgements
	brsmemset(ADR(messages.Read[0]),0,SIZEOF(messages.Read));

END_FUNCTION_BLOCK
```

#### SupertrackPrmyFullBdyInxUnTrack.st
```iecst
(* TODO: Add your comment here *)
FUNCTION_BLOCK SupertrackPrmyFullBdyInxUnTrack

	messages ACCESS p_messages;

	// Debounce Inputs
	DBNC_front_timer(IN := front_raw, PT := DBNC_front_time);
	front := DBNC_front_timer.Q;

	DBNC_after_timer(IN := after_raw, PT := DBNC_after_time);
	after := DBNC_after_timer.Q;

	DBNC_in_pos_timer(IN := in_pos_raw, PT := (DBNC_in_pos_time*2));
	in_pos := DBNC_in_pos_timer.Q;

	ton_lineFull(IN:= full_sensor, PT:= lineFullTime);
	full :=  ton_lineFull.Q;

	// Device State Machine
	IF reset THEN
		udp_data.state := state := ReadyToRelease;
	END_IF;
	IF udp_data.state = 0 THEN udp_data.state := state := ReadyToRelease; END_IF;

	CASE udp_data.state OF
		ReadyToRelease:
			IF fire_os THEN
				udp_data.state := state := Seperate;
			END_IF;

		Seperate:
			IF DBNC_in_pos_timer.Q THEN
				udp_data.state := state := Releasing;
			END_IF;

		Releasing:
			IF after OR NOT(fire) THEN
				udp_data.state := state := ReadyToRelease;
			END_IF;

	END_CASE;

	// Comm Logic
	udp_data.waiting := waiting := (
	udp_data.state = ReadyToRelease
	AND front
	AND NOT(custom_send_lock)
	AND NOT(after)
	AND NOT(safety_zone)
	);

	udp_data.bring_ok := bring_ok := (
	NOT(arrive)
	AND NOT(going_to)
	AND NOT(custom_bring_lock)
	AND NOT(full)
	);

	tof_arrive_dbnc(IN:= EDGENEG(arrive_raw), PT:= dnbc_arrive_time);
	arrive := arrive_raw AND NOT tof_arrive_dbnc.Q;

	IF going_to AND arrive THEN insert := TRUE; END_IF;

	// Output Control
	inx := udp_data.state = Seperate;

	// Pressure Relief
	tof_pressure_1(IN := pressure_full_line_1, PT:= tof_pressureTime);
	pressure_stop_1 := NOT tof_pressure_1.Q;

	tof_pressure_2(IN := pressure_full_line_2, PT:= tof_pressureTime);
	pressure_stop_2 := NOT tof_pressure_2.Q;

	tof_pressure_3(IN := pressure_full_line_3, PT:= tof_pressureTime);
	pressure_stop_3 := NOT tof_pressure_3.Q;

	// Alarm Timers
	AlarmTimer(IN := fire, PT := (t#1s * rail_alarm_time));
	UnexpectedBagTimer(IN := (arrive AND NOT(front) AND NOT(inx)), PT := UnexpectedBagTime);

	// Alarm Coms
	udp_data.alarm := alarm := AlarmTimer.Q;
	udp_data.warning_com.0 := warning_com.0 := UnexpectedBagTimer.Q;

	//Rail Messages
	messages.Write := 0;
	//BAG_STUCK # not yet implemented
	IF UnexpectedBagTimer.Q THEN messages.Write := BIT_SET(messages.Write,UNEXPECTED_BAG); END_IF;

	// Always clear acknowledgements
	brsmemset(ADR(messages.Read[0]),0,SIZEOF(messages.Read));

END_FUNCTION_BLOCK
```

#### SupertrackPrmyFullBdyInxTrack.st
```iecst
(* TODO: Add your comment here *)
FUNCTION_BLOCK SupertrackPrmyFullBdyInxTrack

	messages ACCESS p_messages;

	// Debounce Inputs
	DBNC_front_timer(IN := front_raw, PT := DBNC_front_time);
	front := DBNC_front_timer.Q;

	DBNC_after_timer(IN := after_raw, PT := DBNC_after_time);
	after := DBNC_after_timer.Q;

	DBNC_in_pos_timer(IN := in_pos_raw, PT := (DBNC_in_pos_time*2));
	in_pos := DBNC_in_pos_timer.Q;

	ton_lineFull(IN:= full_sensor, PT:= lineFullTime);
	full :=  ton_lineFull.Q;

	// Device State Machine
	IF reset THEN
		udp_data.state := state := ReadyToRelease;
	END_IF;
	IF udp_data.state = 0 THEN udp_data.state := state := ReadyToRelease; END_IF;

	CASE udp_data.state OF
		ReadyToRelease:
			IF fire_os THEN
				udp_data.state := state := Seperate;
			END_IF;

		Seperate:
			IF DBNC_in_pos_timer.Q THEN
				udp_data.state := state := Releasing;
			END_IF;

		Releasing:
			IF after OR NOT(fire) THEN
				udp_data.state := state := ReadyToRelease;
			END_IF;

	END_CASE;

	// Comm Logic
	udp_data.waiting := waiting := (
	udp_data.state = ReadyToRelease
	AND front
	AND NOT(custom_send_lock)
	AND NOT(after)
	AND NOT(safety_zone)
	);

	udp_data.bring_ok := bring_ok := (
	NOT(arrive)
	AND NOT(going_to)
	AND NOT(custom_bring_lock)
	AND NOT(full)
	);

	tof_arrive_dbnc(IN:= EDGENEG(arrive_raw), PT:= dnbc_arrive_time);
	arrive := arrive_raw AND NOT tof_arrive_dbnc.Q;

	IF going_to AND arrive THEN insert := TRUE; END_IF;

	// Output Control
	inx := udp_data.state = Seperate;

	// Pressure Relief
	tof_pressure_1(IN := pressure_full_line_1, PT:= tof_pressureTime);
	pressure_stop_1 := NOT tof_pressure_1.Q;

	tof_pressure_2(IN := pressure_full_line_2, PT:= tof_pressureTime);
	pressure_stop_2 := NOT tof_pressure_2.Q;

	tof_pressure_3(IN := pressure_full_line_3, PT:= tof_pressureTime);
	pressure_stop_3 := NOT tof_pressure_3.Q;

	// Alarm Timers
	AlarmTimer(IN := fire, PT := (t#1s * rail_alarm_time));
	UnexpectedBagTimer(IN := (arrive AND NOT(front) AND NOT(inx)), PT := UnexpectedBagTime);
	MissingBagTimer(IN := (NOT(front) AND NOT(rail_mt) AND NOT(inx)), PT := MissingBagTime);

	// Alarm Coms
	udp_data.alarm := alarm := AlarmTimer.Q;
	udp_data.warning_com.0 := warning_com.0 := UnexpectedBagTimer.Q;
	udp_data.warning_com.0 := warning_com.0 := MissingBagTimer.Q;

	//Rail Messages
	messages.Write := 0;
	//BAG_STUCK # not yet implemented
	IF UnexpectedBagTimer.Q THEN messages.Write := BIT_SET(messages.Write,UNEXPECTED_BAG); END_IF;
	IF MissingBagTimer.Q THEN messages.Write := BIT_SET(messages.Write,MISSING_BAG); END_IF;

	// Always clear acknowledgements
	brsmemset(ADR(messages.Read[0]),0,SIZEOF(messages.Read));

END_FUNCTION_BLOCK
```

#### SupertrackPrmyHalfBdyInxTrack.st
```iecst
(* TODO: Add your comment here *)
FUNCTION_BLOCK SupertrackPrmyHalfBdyInxTrack

	messages ACCESS p_messages;

	// Debounce Inputs
	DBNC_front_timer(IN := front_raw, PT := DBNC_front_time);
	front := DBNC_front_timer.Q;

	DBNC_after_timer(IN := after_raw, PT := DBNC_after_time);
	after := DBNC_after_timer.Q;

	// Device State Machine
	IF reset THEN
		udp_data.state := state := ReadyToRelease;
	END_IF;
	IF udp_data.state = 0 THEN udp_data.state := state := ReadyToRelease; END_IF;

	CASE udp_data.state OF
		ReadyToRelease:
			IF fire_os THEN
				udp_data.state := state := OpenStop;
			END_IF;

		OpenStop:
			IF ton_open.Q THEN
				udp_data.state := state := Releasing;
			END_IF;

		Releasing:
			IF after OR NOT(fire) THEN
				udp_data.state := state := ReadyToRelease;
			END_IF;

	END_CASE;

	// Comm Logic
	udp_data.waiting := waiting := (
	udp_data.state = ReadyToRelease
	AND front
	AND NOT(custom_send_lock)
	AND NOT(after)
	AND NOT(safety_zone)
	);

	udp_data.bring_ok := bring_ok := (
	NOT(arrive)
	AND NOT(going_to)
	AND NOT(custom_bring_lock)
	);

	tof_arrive_dbnc(IN:= EDGENEG(arrive_raw), PT:= dnbc_arrive_time);
	arrive := arrive_raw AND NOT tof_arrive_dbnc.Q;

	IF going_to AND arrive THEN insert := TRUE; END_IF;

	// Output Control
	inx := udp_data.state = OpenStop;

	ton_open(IN:= (udp_data.state = OpenStop),PT:= openTime);

	// Pressure reliefts
	tof_pressure_1(IN := pressure_full_line_1 OR pressure_stop_1 , PT:= prs_wait_time);
	tof_pressure_2(IN := pressure_full_line_2 OR pressure_stop_2 , PT:= prs_wait_time);
	tof_pressure_3(IN := pressure_full_line_3 OR pressure_stop_3 , PT:= prs_wait_time);

	tof_open_pressure_1(IN := pressure_sensor_1 AND NOT tof_pressure_1.Q, PT:= prs_open_time);
	tof_open_pressure_2(IN := pressure_sensor_2 AND NOT tof_pressure_2.Q, PT:= prs_open_time);
	tof_open_pressure_3(IN := pressure_sensor_3 AND NOT tof_pressure_3.Q, PT:= prs_open_time);

	pressure_stop_1 := tof_open_pressure_1.Q;
	pressure_stop_2 := tof_open_pressure_2.Q;
	pressure_stop_3 := tof_open_pressure_3.Q;

	// Alarm Timers
	AlarmTimer(IN := fire, PT := (t#1s * rail_alarm_time));
	UnexpectedBagTimer(IN := (arrive AND NOT(front) AND NOT(inx)), PT := UnexpectedBagTime);
	MissingBagTimer(IN := (NOT(front) AND NOT(rail_mt) AND NOT(inx)), PT := MissingBagTime);

	// Alarm Coms
	udp_data.alarm := alarm := AlarmTimer.Q;
	udp_data.warning_com.0 := warning_com.0 := UnexpectedBagTimer.Q;
	udp_data.warning_com.0 := warning_com.0 := MissingBagTimer.Q;

	//Rail Messages
	messages.Write := 0;
	//BAG_STUCK # not yet implemented
	IF UnexpectedBagTimer.Q THEN messages.Write := BIT_SET(messages.Write,UNEXPECTED_BAG); END_IF;
	IF MissingBagTimer.Q THEN messages.Write := BIT_SET(messages.Write,MISSING_BAG); END_IF;

	// Always clear acknowledgements
	brsmemset(ADR(messages.Read[0]),0,SIZEOF(messages.Read));

END_FUNCTION_BLOCK
```

#### SupertrackPrmyHalfBdyInxUnTrack.st
```iecst
(* TODO: Add your comment here *)
FUNCTION_BLOCK SupertrackPrmyHalfBdyInxUnTrack

	messages ACCESS p_messages;

	// Debounce Inputs
	DBNC_front_timer(IN := front_raw, PT := DBNC_front_time);
	front := DBNC_front_timer.Q;

	DBNC_after_timer(IN := after_raw, PT := DBNC_after_time);
	after := DBNC_after_timer.Q;

	// Device State Machine
	IF reset THEN
		udp_data.state := state := ReadyToRelease;
	END_IF;
	IF udp_data.state = 0 THEN udp_data.state := state := ReadyToRelease; END_IF;

	CASE udp_data.state OF
		ReadyToRelease:
			IF fire_os THEN
				udp_data.state := state := OpenStop;
			END_IF;

		OpenStop:
			IF ton_open.Q THEN
				udp_data.state := state := Releasing;
			END_IF;

		Releasing:
			IF after OR NOT(fire) THEN
				udp_data.state := state := ReadyToRelease;
			END_IF;

	END_CASE;

	// Comm Logic
	udp_data.waiting := waiting := (
	udp_data.state = ReadyToRelease
	AND front
	AND NOT(custom_send_lock)
	AND NOT(after)
	AND NOT(safety_zone)
	);

	udp_data.bring_ok := bring_ok := (
	NOT(arrive)
	AND NOT(going_to)
	AND NOT(custom_bring_lock)
	);

	tof_arrive_dbnc(IN:= EDGENEG(arrive_raw), PT:= dnbc_arrive_time);
	arrive := arrive_raw AND NOT tof_arrive_dbnc.Q;

	IF going_to AND arrive THEN insert := TRUE; END_IF;

	// Output Control
	inx := udp_data.state = OpenStop;

	ton_open(IN:= (udp_data.state = OpenStop),PT:= openTime);

	// Pressure reliefts
	tof_pressure_1(IN := pressure_full_line_1 OR pressure_stop_1 , PT:= prs_wait_time);
	tof_pressure_2(IN := pressure_full_line_2 OR pressure_stop_2 , PT:= prs_wait_time);
	tof_pressure_3(IN := pressure_full_line_3 OR pressure_stop_3 , PT:= prs_wait_time);

	tof_open_pressure_1(IN := pressure_sensor_1 AND NOT tof_pressure_1.Q, PT:= prs_open_time);
	tof_open_pressure_2(IN := pressure_sensor_2 AND NOT tof_pressure_2.Q, PT:= prs_open_time);
	tof_open_pressure_3(IN := pressure_sensor_3 AND NOT tof_pressure_3.Q, PT:= prs_open_time);

	pressure_stop_1 := tof_open_pressure_1.Q;
	pressure_stop_2 := tof_open_pressure_2.Q;
	pressure_stop_3 := tof_open_pressure_3.Q;

	// Alarm Timers
	AlarmTimer(IN := fire, PT := (t#1s * rail_alarm_time));
	UnexpectedBagTimer(IN := (arrive AND NOT(front) AND NOT(inx)), PT := UnexpectedBagTime);

	// Alarm Coms
	udp_data.alarm := alarm := AlarmTimer.Q;
	udp_data.warning_com.0 := warning_com.0 := UnexpectedBagTimer.Q;

	//Rail Messages
	messages.Write := 0;
	//BAG_STUCK # not yet implemented
	IF UnexpectedBagTimer.Q THEN messages.Write := BIT_SET(messages.Write,UNEXPECTED_BAG); END_IF;

	// Always clear acknowledgements
	brsmemset(ADR(messages.Read[0]),0,SIZEOF(messages.Read));

END_FUNCTION_BLOCK
```

#### SupertrackPrimaryIncline.st
```iecst
(* TODO: Add your comment here *)
FUNCTION_BLOCK SupertrackPrimaryIncline

	messages ACCESS p_messages;

	// Debounce Inputs
	DBNC_after_timer(IN := after_raw, PT := DBNC_after_time);
	after := DBNC_after_timer.Q;

	DBNC_before_timer(IN := before_raw, PT := DBNC_before_time);
	before := DBNC_before_timer.Q;

	//debounce timer for top sensor as the bag can swing when releasing
	ton_top_sensor_dnbc(IN:=(udp_data.state = Releasing) AND conveyor_running, PT:= dbnc_top_switch_time);
	//Clear the trolley at top bit when we have released the trolley from the inclines.
	IF ton_top_sensor_dnbc.Q THEN
		trolleyAtTop := 0;
	END_IF;

	//Detect the EDGE of the trolley moving off the out sensor
	IF EDGEPOS(rail_out_sensor) THEN
		trolleyAtTop := 1;
	END_IF;

	// Move this outside the case so that we can see the edge correctly
	IF  EDGEPOS(trolleyAtTop) AND (udp_data.state = Releasing)  THEN
		udp_data.state := state := ReadyToRelease;
	END_IF;

	// Device State Machine
	IF reset THEN
		udp_data.state := state := ReadyToWork;
		IF rail_mt THEN
			trolleyAtTop := 0;
		END_IF;
	END_IF;
	IF udp_data.state = 0 THEN udp_data.state := state := ReadyToWork; END_IF;

	CASE udp_data.state OF

		ReadyToWork: // Motor can run  if not MT
			IF trolleyAtTop THEN
				udp_data.state := state := ReadyToRelease;
			ELSIF before AND NOT rail_full THEN
				udp_data.state := state := AlignLift;
			END_IF;

		AlignLift: // Find the paddle in position
			IF trolleyAtTop THEN
				udp_data.state := state := ReadyToRelease;
			ELSIF rail_full THEN
				udp_data.state := state := ReadyToWork;
			ELSIF paddle_sensor THEN
				udp_data.state := state := Receiving;
			END_IF;

		Receiving: // Motor stopped and bag coming in from buffer
			IF arrive_raw THEN
				udp_data.state := state := ReadyToWork;
			END_IF;

		ReadyToRelease:
			IF fire_os THEN
				udp_data.state := state := Releasing;
			END_IF;

		Releasing:
			IF after OR NOT(fire)  THEN
				trolleyAtTop := 0;
				udp_data.state := state := ReadyToWork;
			ELSIF NOT trolleyAtTop AND before AND NOT rail_full AND NOT rail_mt AND paddle_sensor  THEN
				udp_data.state := state := Receiving;
			END_IF;

	END_CASE;

	// Comm Logic
	udp_data.waiting := waiting := (
	udp_data.state = ReadyToRelease
	AND NOT(custom_send_lock)
	AND NOT(after)
	AND NOT(safety_zone)
	);

	udp_data.bring_ok := bring_ok := (
	NOT(arrive)
	AND NOT(going_to)
	AND NOT(custom_bring_lock)
	AND (udp_data.state = Receiving)
	);

	arrive := arrive_raw;

	IF going_to AND arrive THEN insert := TRUE; END_IF;

	// Output Control;
	run_slant := (
	(((((udp_data.state = ReadyToWork) AND (NOT rail_mt OR (fire AND rail_mt))) OR (udp_data.state = AlignLift)) AND NOT trolleyAtTop)
	OR (udp_data.state = Releasing))
	AND onoff
	);

	// Alarm Timers
	AlarmTimer(IN := fire, PT := (t#1s * rail_alarm_time));
	UnexpectedBagTimer(IN := (arrive AND rail_mt AND NOT(run_slant)), PT := UnexpectedBagTime);

	// Alarm Coms
	udp_data.alarm := alarm := AlarmTimer.Q;
	udp_data.warning_com.0 := warning_com.0 := UnexpectedBagTimer.Q;

	messages.Write := 0;
	IF UnexpectedBagTimer.Q   THEN messages.Write := BIT_SET(messages.Write,UNEXPECTED_BAG); END_IF;

	// Always clear acknowledgements
	brsmemset(ADR(messages.Read[0]),0,SIZEOF(messages.Read));

END_FUNCTION_BLOCK
```

#### SupertrackPrimaryUnLoadingPoint.st
```iecst
(* TODO: Add your comment here *)
FUNCTION_BLOCK SupertrackPrimaryUnLoadingPoint

	messages ACCESS p_messages;

	// Debounce Inputs
	DBNC_front_timer(IN := front_raw, PT := DBNC_front_time);
	front := DBNC_front_timer.Q;

	// Device State Machine
	IF reset THEN
		IF front THEN
			udp_data.state := state := ReadyToUnload;
		ELSE
			udp_data.state := state := ReadyToWork;
		END_IF;
	END_IF;

	IF udp_data.state = 0 THEN udp_data.state := state := ReadyToWork; END_IF;

	CASE udp_data.state OF

		ReadyToWork:
			IF front AND onoff AND NOT(halted) THEN
				udp_data.state := state := ReadyToUnload;
			END_IF;

		ReadyToUnload:
			IF man_send OR EDGENEG(foot) THEN
				man_send := 0;
				udp_data.state := state := ReadyToRelease;
			END_IF;

		ReadyToRelease:
			IF fire_os THEN
				udp_data.state := state := Releasing;
			END_IF;

		Releasing:
			IF NOT(fire) OR after THEN
				udp_data.state := state := ReadyToWork;
			END_IF;

	END_CASE;

	// Comm Logic
	udp_data.waiting := waiting := (
	udp_data.state = ReadyToRelease
	AND NOT(custom_send_lock)
	AND NOT(after)
	AND NOT(safety_zone)
	);

	udp_data.bring_ok := bring_ok := (
	udp_data.state = ReadyToWork
	AND NOT(arrive)
	AND NOT(front)
	AND NOT(going_to)
	AND NOT(custom_bring_lock)
	);

	IF going_to AND arrive THEN insert := TRUE; END_IF;

	// Input Control
	arrive := arrive_raw := front_raw;
	after := after_raw;

	// Output Control
	stp := (udp_data.state = Releasing);

	// Alarm Timers
	AlarmTimer(IN := fire, PT := (t#1s * rail_alarm_time));
	UnexpectedBagTimer(IN := (front AND rail_mt), PT := UnexpectedBagTime);

	// Alarm Coms
	udp_data.alarm := alarm := AlarmTimer.Q;
	udp_data.warning_com.0 := warning_com.0 := UnexpectedBagTimer.Q;

	//Rail Messages
	messages.Write := 0;
	//BAG_STUCK # not yet implemented
	IF UnexpectedBagTimer.Q THEN messages.Write := BIT_SET(messages.Write,UNEXPECTED_BAG); END_IF;

	// Always clear acknowledgements
	brsmemset(ADR(messages.Read[0]),0,SIZEOF(messages.Read));

END_FUNCTION_BLOCK
```

#### SupertrackPrimaryBagRemover.st
```iecst
(* TODO: Add your comment here *)
FUNCTION_BLOCK SupertrackPrimaryBagRemover

	messages ACCESS p_messages;

	// Debounce Inputs
	DBNC_front_timer(IN := front_raw, PT := DBNC_front_time);
	front := DBNC_front_timer.Q;

	DBNC_after_timer(IN := after_raw, PT := DBNC_after_time);
	after := DBNC_after_timer.Q;

	// Device State Machine
	IF reset THEN udp_data.state := state := ReadyToWork; END_IF;
	IF udp_data.state = 0 THEN udp_data.state := state := ReadyToWork; END_IF;

	CASE udp_data.state OF

		ReadyToWork:
			IF (front_raw OR going_to) AND onoff AND NOT(halted) THEN
				udp_data.state := state := Receiving;
			END_IF;

		Receiving:
			IF front THEN
				udp_data.state := state := StripBag;
			END_IF;

		StripBag:
			IF ton_strip.Q THEN
				udp_data.state := state := ReadyToRelease;
			END_IF;

		ReadyToRelease:
			IF fire THEN //(Use the .fire not the edge, so we can retry on a timeout.)
				udp_data.state := state := Releasing;
			END_IF;

		Releasing:
			IF NOT(fire) OR after THEN
				udp_data.state := state := ReadyToWork;
			ELSIF ton_timeout.Q THEN
				udp_data.state := state := StripBag;
			END_IF;

	END_CASE;

	// Comm Logic
	udp_data.waiting := waiting := (
	udp_data.state = ReadyToRelease
	AND front
	AND NOT(custom_send_lock)
	AND NOT(after_raw)
	AND NOT(safety_zone)
	);

	udp_data.bring_ok := bring_ok := (
	udp_data.state = ReadyToWork
	AND NOT(front_raw)
	AND NOT(custom_bring_lock)
	AND NOT(safety_zone)
	);

	IF going_to AND arrive THEN insert := TRUE; END_IF;

	// Input Control
	arrive := arrive_raw := front_raw;

	// Output Control
	stp := (udp_data.state = Releasing);

	grab := ((udp_data.state = ReadyToRelease) OR (udp_data.state = StripBag));

	ton_timeout(IN:= (udp_data.state = Releasing), PT:= releaseTime);
	ton_strip(IN:= (udp_data.state = StripBag), PT:= stripTime);

	// Alarm Timers
	AlarmTimer(IN := fire, PT := (t#1s * rail_alarm_time));

	// Alarm Coms
	udp_data.alarm := alarm := AlarmTimer.Q;

	//Rail Messages
	messages.Write := 0;
	//BAG_STUCK # not yet implemented
	//IF UnexpectedBagTimer.Q THEN messages.Write := BIT_SET(messages.Write,UNEXPECTED_BAG); END_IF;

	// Always clear acknowledgements
	brsmemset(ADR(messages.Read[0]),0,SIZEOF(messages.Read));

END_FUNCTION_BLOCK
```

#### SupertrackRudderStp.st
```iecst
(* TODO: Add your comment here *)
FUNCTION_BLOCK SupertrackRudderStp

	messages ACCESS p_messages;

	  // Debounce Inputs
	DBNC_front_timer(IN := front_raw, PT := DBNC_front_time);
	front := DBNC_front_timer.Q;

	DBNC_arrive_timer(IN := arrive_raw, PT := DBNC_arrive_time);
	arrive := DBNC_arrive_timer.Q;

	DBNC_after_timer(IN := after_raw, PT := DBNC_after_time);
	after := DBNC_after_timer.Q;

	DBNC_before_timer(IN := before_raw, PT := DBNC_before_time);
	before := DBNC_before_timer.Q;

	DBNC_after_a_timer(IN := after_a_raw, PT := DBNC_after_a_time);
	after_a := DBNC_after_a_timer.Q;

	DBNC_after_b_timer(IN := after_b_raw, PT := DBNC_after_b_time);
	after_b := DBNC_after_b_timer.Q;

	// Device State Machine
	IF reset THEN udp_data.state := state := ReadyToWork; END_IF;
	IF udp_data.state = 0 THEN
		udp_data.state := state := ReadyToWork;;
		front_a_seen := FALSE;
	END_IF;

	CASE udp_data.state OF
		ReadyToWork:
			IF front_a AND NOT(front_a_seen) THEN
				front_a_seen := TRUE;
			ELSIF NOT(rail_mt) AND front AND onoff AND NOT(halted) THEN
				udp_data.state := state := ReadyToRelease;
			END_IF;

		ReadyToRelease:
			IF fire_os THEN
				udp_data.state := state := ReleasingFront;
				front_a_seen := FALSE;
			END_IF;

		ReleasingFront:
			IF after_a THEN
				udp_data.state := state := ReleasingRear;
			ELSIF NOT(fire) OR after THEN
				udp_data.state := state := ReadyToWork;
			END_IF;

		ReleasingRear:
			IF after_b OR NOT(fire) THEN
				udp_data.state := state := ReadyToWork;
			END_IF;

	END_CASE;

	// Comm Logic
	udp_data.waiting := waiting := (
	udp_data.state = ReadyToRelease
	AND front
	AND NOT(custom_send_lock)
	AND NOT(after_b)
	AND NOT(after)
	AND NOT(safety_zone)
	);

	udp_data.bring_ok := bring_ok := (
	udp_data.state = ReadyToWork
	AND NOT(going_to)
	AND NOT(before)
	AND NOT(arrive)
	AND NOT(front_a)
	AND NOT(front_b)
	AND NOT(custom_bring_lock)
	);

	IF going_to AND arrive THEN insert := TRUE; END_IF;

	// Input Control
	arrive_raw := front_raw := front_a_seen AND front_b;

	// Output Control
	stp := udp_data.state = ReleasingFront OR udp_data.state = ReleasingRear;
	stp_a := udp_data.state = ReleasingFront OR udp_data.state = ReleasingRear;
	stp_b := udp_data.state = ReleasingRear;

	// Output Switch Control
	IF SwInARTrig.Q THEN
		sw_in_a := TRUE;
	END_IF;

	IF before AND going_to THEN
		sw_in_a := FALSE;
		sw_in_b  := TRUE;
	END_IF;

	IF NOT(going_to) THEN
		sw_in_a := FALSE;
		sw_in_b  := FALSE;
	END_IF;

	IF SwOutARTrig.Q THEN
		sw_out_a := TRUE;
	END_IF;

	IF fire AND after THEN
		sw_out_a := FALSE;
		sw_out_b  := TRUE;
	END_IF;

	IF NOT(fire) THEN
		sw_out_a := FALSE;
		sw_out_b  := FALSE;
	END_IF;

	IF reset THEN
		sw_out_a := FALSE;
		sw_out_b  := FALSE;
	END_IF;

	// Control Triggers
	SwInARTrig(CLK := (going_to));
	SwOutARTrig(CLK := (fire));

	// Alarm Timers
	AlarmTimer(IN := fire, PT := (t#1s * rail_alarm_time));
	UnexpectedBagTimer(IN := (front AND rail_mt), PT := UnexpectedBagTime);
	MissingBagTimer(IN := (NOT(front) AND NOT(rail_mt)), PT := MissingBagTime);

	// Alarm Coms
	udp_data.alarm := alarm := AlarmTimer.Q;
	udp_data.warning_com.0 := warning_com.0 := UnexpectedBagTimer.Q;
	udp_data.warning_com.1 := warning_com.1 := MissingBagTimer.Q;

	messages.Write := 0;
	IF UnexpectedBagTimer.Q   THEN messages.Write := BIT_SET(messages.Write,UNEXPECTED_BAG); END_IF;
	IF MissingBagTimer.Q      THEN messages.Write := BIT_SET(messages.Write,MISSING_BAG); END_IF;

	// Always clear acknowledgements
	brsmemset(ADR(messages.Read[0]),0,SIZEOF(messages.Read));

END_FUNCTION_BLOCK
```

### Safety.typ
```iecst
TYPE
	SafeTowerLightType : 	STRUCT
		TL_DO_Green : BOOL; (*Tower light output for Green light*)
		TL_DO_Yellow : BOOL; (*Tower light output for Yellow light*)
		TL_DO_Red : BOOL; (*Tower light output for Red light*)
		TL_DO_Sounder : BOOL; (*Tower light output for sounder*)
	END_STRUCT;
	SafeZoneType : 	STRUCT
		TowerLight : SafeTowerLightType; (*Tower light structure*)
		AccessRequested : BOOL; (*Operator as requested access*)
		RequestAccess : BOOL; (*Command to request Access ON with Reset PB and Zone Status is Healthy.*)
		Main_Lamp : BOOL; (*Main panel lamp*)
		BagsInTransit : BOOL; (*True = Sequences are still not in a safe step*)
		HoistsOutOfPosition : BOOL; (*True = Hoists in zone are not parked*)
		Disable : BOOL; (*Passed into sequences to inhibit stepping on*)
		EDM : BOOL; (*EDM Feedback from linking relays*)
		ResetReady : BOOL; (*Zone is ready to be reset*)
		LiftGates : BOOL; (*Lift the edge protection gates.*)
		HaltSys : BOOL;
		Zone_Status : BOOL; (*State of the zone passed back from safe PLC*)
		PressureSwitch : BOOL;
		DoorLock : BOOL; (**Lock Doors in the area*)
		SafeInput : BOOL; (**Safety Input Condition Passed from Safe PLC*)
		ResetButton : BOOL;
		DataFromSafePLC : INT; (*Data from Safety PLC*)
	END_STRUCT;
	Safety_Hoist_type : 	STRUCT
		O_OpenGuard : BOOL; (*Sliding guard output*)
		O_CloseGuard : BOOL; (*Sliding guard output*)
		OutOfPosition : BOOL; (*True when hoist is not in Service position*)
	END_STRUCT;
	Safety_typ : 	STRUCT
		ModuleOk : BOOL;
		ModuleID : UDINT;
		FW_Version : UDINT;
		SFW_Version : UINT;
		UDID_low : UDINT;
		UDID_high : UINT;
		ModuleFault : BOOL;
		MasterReset_Comm : INT; (**Bits to do a master reset on a collection of safety zones*)
		EDM_Comm : DINT; (**EDM states packed for PLC comm*)
		Reset_Comm : DINT; (**Bits to reset zone with no reset button accessible via SD*)
	END_STRUCT;
	SM_type : 	STRUCT  (**Safety Module type*)
		ModuleOk : BOOL;
		SerialNumber : UDINT;
		ModuleID : UINT;
		HardwareVariant : UINT;
		FirmwareVersion : UINT;
		SafeModuleOK : BOOL;
		SafeDigitialInput01 : BOOL;
		SafeDigitialInput02 : BOOL;
		SafeDigitialInput03 : BOOL;
		SafeDigitialInput04 : BOOL;
		SafeDigitialInput05 : BOOL;
		SafeDigitialInput06 : BOOL;
		SafeDigitialInput07 : BOOL;
		SafeDigitialInput08 : BOOL;
		SafeTwoChannelInput0102 : BOOL;
		SafeTwoChannelInput0304 : BOOL;
		SafeTwoChannelInput0506 : BOOL;
		SafeTwoChannelInput0708 : BOOL;
		SafeTwoChannelOk0102 : BOOL;
		SafeTwoChannelOk0304 : BOOL;
		SafeTwoChannelOk0506 : BOOL;
		SafeTwoChannelOk0708 : BOOL;
		DigitalInput01 : BOOL;
		DigitalInput02 : BOOL;
		DigitalOutput01 : BOOL;
		DigitalOutput02 : BOOL;
	END_STRUCT;
END_TYPE
```

### Safety.var
```iecst
VAR
	SM : ARRAY[0..3999] OF SM_type;
	SafetyZone : ARRAY[0..MAX_SAFE_ZONES] OF SafeZoneType;
	Hoist_Safety : ARRAY[0..MAX_HOIST] OF Safety_Hoist_type;
	Safety : Safety_typ;
END_VAR
```

### Program Logical/Safety/AccessControl (IEC) - *Mapping to allow access into zones

#### Main.st
```iecst
PROGRAM _CYCLIC

//	Std.SafetyOnZone[1]	;Soiled EStops + SIC1-4 + SIC7
//	Std.SafetyOnZone[2]	;SSL1 Guarded Area + STB1, STB2, STB11
//	Std.SafetyOnZone[3]	;SSL2 Guarded Area + STB3, STB4, STB12
//	Std.SafetyOnZone[4]	;STB5, STB6, STB7
//	Std.SafetyOnZone[5]	;STB8, STB9, STB10
//	Std.SafetyOnZone[6]	;SB1
//	Std.SafetyOnZone[7]	;SB2
//	Std.SafetyOnZone[8]	;SB3
//	Std.SafetyOnZone[9]	;SB4
//
//No access on zone 0

	//	SafetyZone[0].BagsInTransit :=  FALSE;  // Safe to enter when false (Switch is NO) FALSE WHEN OK..
	//	SafetyZone[0].HoistsOutOfPosition := FALSE; //<-- This is used to stop the door from opening if not position FALSE IS OK -- SWITCH IS NC..
	SafetyZone[1].ResetButton := X[1001].X03 OR X[1003].X03;
	SafetyZone[2].ResetButton := SM[1401].DigitalInput01 OR SM[1404].DigitalInput01;
	SafetyZone[3].ResetButton := SM[1402].DigitalInput01 OR SM[1406].DigitalInput01;
	SafetyZone[4].ResetButton := SM[1402].DigitalInput02;
	SafetyZone[5].ResetButton := SM[1406].DigitalInput02;
	SafetyZone[6].ResetButton := X[1001].X03 OR X[1003].X03;
	SafetyZone[7].ResetButton := X[1001].X03 OR X[1003].X03;
	SafetyZone[8].ResetButton := X[1001].X03 OR X[1003].X03;
	SafetyZone[9].ResetButton := X[1001].X03 OR X[1003].X03;

	SafetyZone[1].BagsInTransit :=  FALSE;
	SafetyZone[1].HoistsOutOfPosition := FALSE;

	SafetyZone[2].BagsInTransit :=  FALSE;
	SafetyZone[2].HoistsOutOfPosition := FALSE;

	SafetyZone[3].BagsInTransit :=  FALSE;
	SafetyZone[3].HoistsOutOfPosition := FALSE;

	SafetyZone[4].BagsInTransit :=  FALSE;
	SafetyZone[4].HoistsOutOfPosition := FALSE;

	SafetyZone[5].BagsInTransit :=  FALSE;
	SafetyZone[5].HoistsOutOfPosition := FALSE;

	SafetyZone[6].BagsInTransit :=  FALSE;
	SafetyZone[6].HoistsOutOfPosition := FALSE;

	SafetyZone[7].BagsInTransit :=  FALSE;
	SafetyZone[7].HoistsOutOfPosition := FALSE;

	SafetyZone[8].BagsInTransit :=  FALSE;
	SafetyZone[8].HoistsOutOfPosition := FALSE;

	SafetyZone[9].BagsInTransit :=  FALSE;
	SafetyZone[9].HoistsOutOfPosition := FALSE;

	SM[1401].DigitalOutput01 := SafetyZone[2].DoorLock; //SSL1,STB1,STB2,STB11
	SM[1402].DigitalOutput01 := SafetyZone[3].DoorLock; //SSL2,STB3,STB4,STB12
	//SM[1403].DigitalOutput01 := SafetyZone[10].DoorLock; //SSL3
	SM[1404].DigitalOutput01 := SafetyZone[2].DoorLock; //SSL1,STB1,STB2,STB11
	SM[1404].DigitalOutput02 := SafetyZone[4].DoorLock; //STB5,STB6,STB7
	SM[1406].DigitalOutput01 := SafetyZone[3].DoorLock; //SSL2,STB3,STB4,STB12
	SM[1406].DigitalOutput02 := SafetyZone[13].DoorLock; //STB8,STB9,STB10

END_PROGRAM
```

### Program Logical/Safety/Safety (IEC, version 2.00.1)

#### Main.st - Safet Task must come after all task with gaurded areas
```iecst
//---------------------------------------------
//-------------Safety Request------------------
//---------------------------------------------
//V1.00.2 -- 2019 May 24 -- TR -- Fix issue with master reset not working if not ready.
//V1.00.3 -- 2019 June 26 -- TR -- FIx issue with the solenoid not opening if the hoist switch is made after the bagInTransit timers.. Add timer for hoist in position so the hoist cannot be moving past the safe position and open the door.
//V1.00.4 -- 2019 November 11 -- TR -- 	FIX: Issues with the solenoid locking incorrectly,
						//ADD: Control to lift the edge protection gates ( Map Directly to all required outputs.)
//V1.00.5 -- 2020 Decemeber 16 -- TR -- UPDATE : Change to new structure for Safety.
//V1.00.6 -- 2021 January 02 -- TR -- UPDATE : Add Test Mode bit
//V2.00.1 - 2001 Feburary 05 - Change Structures to remove links to direct IO points. Data now comes from Safe PLC.

PROGRAM _INIT

//***************************************************************************************
//	N.B Zone 11 has been faked so we can control the lamp tower correctly FOR the primary
//***************************************************************************************

//DECLARE MAX_SAFE_SYSTEMS IN CONTSTANTS

	startZone[1] := 1;   // Number of the Master Zone
	endZone[1] := 5;	// Last zone in the area
	enableMasterReset[1] := TRUE; // Set to true if master reset is to be used/
//	alarmCondition[1] := system_alarm_1 OR soiled_validation_alarm OR halted;

	//zone for clean alarms.
	startZone[2] := 11;   // Number of the Master Zone
	endZone[2] := MAX_SAFE_ZONES;	// Last zone in the area
	enableMasterReset[2] := TRUE; // Set to true if master reset is to be used/

	//NB//  A ZONE CANNOT BELONG TO MORE THAN 1 SAFE SYSTEM.

	// MAX Zone if 30

	debounceMasterPT := 476; //4.76 second
	transitSettlePT := 3000; //3000seconds
	startUpWarningPT := 500; //5 secs

	FOR n:=1 TO MAX_SAFE_ZONES DO
		safeState[n] := 4;
	END_FOR;

	#if (MAX_SAFE_ZONES  > 30)
	#error 'Cannot have more than 30 safety zones'
	#endif

END_PROGRAM

PROGRAM _CYCLIC

alarmCondition[1] := system_alarm_1 OR soiled_validation_alarm OR halted;
alarmCondition[2] := system_alarm_2 OR clean_validation_alarm OR halted;

FOR s := 1 TO MAX_SAFE_SYSTEMS DO

	ton_10ms_startUp_Warning[s].IN:= masterResetRequest[s];
	ton_10ms_startUp_Warning[s].PT:= startUpWarningPT;
	ton_10ms_startUp_Warning[s]();

	IF  ton_10ms_startUp_Warning[s].Q AND Std.Clock1s THEN
		Safety.MasterReset_Comm	:= BIT_SET(Safety.MasterReset_Comm,s);
	ELSE
		Safety.MasterReset_Comm	:= BIT_CLR(Safety.MasterReset_Comm,s);
	END_IF;

	masterZoneNo := startZone[s]; // Number of the master zone for the safe system.

	ton_10ms_Master_Reset[s].IN:= SafetyZone[masterZoneNo].ResetButton AND enableMasterReset[s];//masterResetRequest[s];
	ton_10ms_Master_Reset[s].PT:= debounceMasterPT;
	ton_10ms_Master_Reset[s]();

	IF 	ton_10ms_Master_Reset[s].Q THEN
		masterResetRequest[s] := 1;
	END_IF;

	tmrAlmOutput[s].IN := alarmCondition[s];
	tmrAlmOutput[s].PT := T#5s;
	tmrAlmOutput[s]();

	FOR n:= startZone[s] TO endZone[s] DO

		IF startZone[s] = 0 THEN
			EXIT;
		END_IF;

		safeZone ACCESS ADR(SafetyZone[n]);
		masterZone := (n = startZone[s]);

		_decodeData;

		//Set the EDM bit//
		IF safeZone.EDM THEN
			Safety.EDM_Comm := BIT_SET(Safety.EDM_Comm,n);
		ELSE
			Safety.EDM_Comm := BIT_CLR(Safety.EDM_Comm,n);
		END_IF;

		//set the reset bit//
		IF safeZone.ResetButton THEN
			Safety.Reset_Comm := BIT_SET(Safety.Reset_Comm,n);
		ELSE
			Safety.Reset_Comm := BIT_CLR(Safety.Reset_Comm,n);
		END_IF;

		//-------------------------------------------------------
		//---------------------Master-reset----------------------
		//-------------------------------------------------------
		IF Std.TestMode AND (Safety.SFW_Version = 0) THEN
			safeZone.DoorLock 	:= FALSE;
			safeZone.LiftGates 	:= FALSE;
			safeZone.Zone_Status 	:= TRUE;
			safeZone.Disable 		:= FALSE;
			safeZone.HaltSys 		:= NOT(safeZone.Zone_Status AND NOT safeZone.Disable);
		ELSE
			lockDoor[n] := FALSE;

			tof_HoistsOutOfPosition[n].IN := safeZone.HoistsOutOfPosition;
			tof_HoistsOutOfPosition[n].PT := 100;
			tof_HoistsOutOfPosition[n]();

			ton_entryError[n].IN := (safeState[n] = 3);
			ton_entryError[n].PT := 100;
			ton_entryError[n]();

			IF ton_10ms_Master_Reset[s].Q AND NOT safeZone.Zone_Status AND safeZone.ResetReady THEN // only put a zone to reset if it needs it
				masterReset[n] := TRUE; // Set masterReset
				safeState[n] := 10; // Goto master reset state
			END_IF;

			//-------------------------------------------------------
			//------------------END-Master-Reset-END-----------------
			//-------------------------------------------------------

			//-------------------------------------------------------
			//------------------Safety-State-Machine-----------------
			//-------------------------------------------------------

			//Wait for bags to finish moving and hoists to get into position.. Door can be unlocked
			ton_10ms_Transit_Settle[n](IN:= safeZone.AccessRequested AND (safeState[n] = 1), PT:=transitSettlePT);
			IF NOT masterZone THEN
				f_trigRequestAccess[n].CLK:= safeZone.RequestAccess;
				f_trigRequestAccess[n]();
			END_IF;
			CASE safeState[n] OF
				0: //Zone reset do not enter

					// Operator requests access by pressing Access DI for 1 second then releasing
					IF safeZone.AccessRequested THEN
						safeState[n] := 1;
					ELSIF safeZone.Zone_Status AND f_trigRequestAccess[n].Q  THEN//	ELSIF (debounceEdgeNeg[n] OR safeZone.AccessRequested) AND NOT masterReset THEN //Look for falling edge if masterReset not requested
						safeZone.AccessRequested := TRUE; //Reset after unlocking or safe zone goes off
						safeState[n] := 1; //Access has been requested
						masterReset[n] := 0;
						//If zone accessed by override or depedant Zone drops out.
					ELSIF NOT safeZone.Zone_Status AND NOT safeZone.SafeInput THEN //If entered with overide goto state 3
						safeState[n] := 3;
					ELSIF NOT safeZone.Zone_Status AND safeZone.SafeInput THEN //If dependant zone drops out
						safeState[n] := 4;
					END_IF;

				1: //Access has been requested
					//Allow 1 second for moving bags to settle, once ok
					ton_10ms_bagsInTransit[n](IN:=NOT safeZone.BagsInTransit, PT:=100); //buffer the BagsInTransit bool

					//Latch solenoid lock open
					IF ton_10ms_bagsInTransit[n].Q AND safeZone.Disable AND NOT tof_HoistsOutOfPosition[n].Q THEN //Use Disable instead of AccessRequested, to ensure one cyclic check with Disable on to stop BagsInTransit being missed
						//safeZone.LockDoors := TRUE; //Reset after reset pressed and door shut
						safeState[n] := 2; //Safe to enter no bags in transit
					ELSIF ton_10ms_Transit_Settle[n].Q THEN
						//safeZone.LockDoors := NOT tof_HoistsOutOfPosition[n].Q; //Reset after reset pressed and door shut
						safeState[n] := 3; //Waiting time elapsed, enter with caution
					END_IF;

					//If zone accessed by override or depedant Zone drops out.
					IF NOT safeZone.Zone_Status AND NOT safeZone.SafeInput THEN //If entered with overide goto state 3
						safeState[n] := 3;
					ELSIF NOT safeZone.Zone_Status AND safeZone.SafeInput THEN //If dependant zone drops out
						safeState[n] := 4;
					ELSIF safeZone.Zone_Status AND f_trigRequestAccess[n].Q THEN //Cancel the request
						safeZone.AccessRequested := FALSE; //Reset after safe zone goes off
						safeState[n] := 4;
					END_IF;

				2..3: //Zone unlocked
					//Reset access request
					lockDoor[n] := NOT tof_HoistsOutOfPosition[n].Q;

					IF safeZone.AccessRequested AND NOT safeZone.Zone_Status THEN
						safeZone.AccessRequested := FALSE; //Reset after safe zone goes off
						IF n = 0 THEN
							safeState[n] := 0; //Zone reset do not enter
						END_IF
					ELSIF safeZone.Zone_Status AND f_trigRequestAccess[n].Q  AND safeZone.AccessRequested THEN //Cancel the request
						safeZone.AccessRequested := FALSE; //Reset after safe zone goes off
						safeState[n] := 4;
					ELSIF safeZone.Zone_Status AND NOT safeZone.AccessRequested THEN // zone has been accessed and reset.
						safeState[n] := 0;
					END_IF;

				4:
					//Reset tower light state only if safety plc feedback ok
					IF safeZone.Zone_Status THEN //Check Safe PLC status
						safeState[n] := 0; //Zone reset do not enter
					END_IF;

				10: // Master reset
					IF (safeZone.Zone_Status OR NOT safeZone.ResetReady) THEN
						safeState[n] := 0;
						masterReset[n] := FALSE;
					END_IF;

			END_CASE;

			//	//Lock solenoid
			//	//ton_10ms_Reset_Debounce[n](IN:=safeZone.Interlock.GS_DI_01_Access_Reset, PT:=debouncePT);
			//	IF (safeZone.Interlock.GS_DI_01_Access_Reset AND (safeState[n] > 1) AND NOT masterReset[n]) THEN
			//		//safeZone.LockDoors := FALSE; //Reset after reset pressed and door shut
			//		safeZone.AccessRequested := FALSE;
			//		safeState[n] := 4; // Check zone status
			//		//		ELSIF masterReset AND NOT safeZone.Zone_Status AND safeZone.ResetReady THEN
			//		//			safeState[n] := 10; // Goto master reset state
			//	END_IF;

			//Set disable to safe zone off or access requested
			safeZone.Disable := safeZone.AccessRequested OR NOT safeZone.Zone_Status;

			//-------------------------------------------------------
			//-------END--------Safety State Machine-------END-------
			//-------------------------------------------------------

			//-------------------------------------------------------
			//---------Set tower light status-&-TV-Indicators--------
			//-------------------------------------------------------
			IF NOT masterZone THEN //Light tower 0 does not need to indicate access state.. It is used on the main cab to indicate alarms. See alarm Task.
				safeZone.TowerLight.TL_DO_Green := safeZone.TowerLight.TL_DO_Yellow := safeZone.TowerLight.TL_DO_Red := safeZone.TowerLight.TL_DO_Sounder := 0;
				CASE safeState[n] OF
					0: //Zone reset do not enter
						safeZone.TowerLight.TL_DO_Green 	:= safeZone.Zone_Status;
						safeZone.TowerLight.TL_DO_Red 		:= NOT safeZone.Zone_Status;
					1: //Access has been requested
						safeZone.TowerLight.TL_DO_Yellow 	:= Std.Clock1s; 	//Means Zone Ok but access requested
						safeZone.TowerLight.TL_DO_Green 	:= safeZone.Zone_Status;
						safeZone.TowerLight.TL_DO_Red 		:= NOT safeZone.Zone_Status;
					2: //Safe to enter no bags in transit and hoists in position
						safeZone.TowerLight.TL_DO_Yellow 	:= TRUE; //Amber & RED steady indicates safe to enter
						safeZone.TowerLight.TL_DO_Green 	:= safeZone.Zone_Status;
						safeZone.TowerLight.TL_DO_Red 		:= TRUE;
					3: //
						safeZone.TowerLight.TL_DO_Yellow 	:= Std.Clock200ms; //Amber/Green Alternate-- Enter with Caution
						safeZone.TowerLight.TL_DO_Sounder 	:= NOT ton_entryError[n].Q; //Short alarm to indicate enter with caution
						safeZone.TowerLight.TL_DO_Green 	:= NOT Std.Clock200ms;
						safeZone.TowerLight.TL_DO_Red 		:= NOT Std.Clock200ms OR safeZone.HoistsOutOfPosition; // If red ight on then fault

					4: //Ready for Reset
						safeZone.TowerLight.TL_DO_Yellow 	:= Std.Clock500ms AND safeZone.ResetReady; //Flash Yellow when ready to be reset
						safeZone.TowerLight.TL_DO_Green 	:= safeZone.Zone_Status;

					10://Master Reset Zone about to start
						safeZone.TowerLight.TL_DO_Sounder := TRUE;
						safeZone.TowerLight.TL_DO_Red := Std.Clock200ms; //Red fast flash indicates zone will reset
				END_CASE;

			ELSE // Master Zone lamp controls
				safeZone.TowerLight.TL_DO_Red 		:= FALSE;
				safeZone.TowerLight.TL_DO_Yellow	:= FALSE;
				safeZone.TowerLight.TL_DO_Green	:= FALSE;

				IF safeZone.HaltSys AND NOT safeZone.ResetReady THEN	//Emergency stop blink red. (State 1)
					safeZone.TowerLight.TL_DO_Red 		:= Std.Clock1s ;
				ELSIF safeZone.HaltSys THEN // Estop waiting for reset  (State 2)
					safeZone.TowerLight.TL_DO_Yellow		:= Std.Clock1s;
				ELSIF alarmCondition[s] THEN //State 10 -- Show Warning Not Fault when alarm is on as other parts might still be running
					safeZone.TowerLight.TL_DO_Yellow 	:= TRUE;
					safeZone.TowerLight.TL_DO_Green	 := TRUE;
				ELSE //Machine Running (State 6)
					safeZone.TowerLight.TL_DO_Green	 := TRUE;
				END_IF;
				safeZone.TowerLight.TL_DO_Sounder := (alarmCondition[s] AND NOT tmrAlmOutput[s].Q);

			END_IF;

			//-------------------------------------------------------------
			//-------END-Set tower light status-&-TV-Indicators-END--------
			//-------------------------------------------------------------

			//Check if the master reset has reset all zones.
			IF (masterReset[n] AND NOT safeZone.Zone_Status) THEN
				resetRequired[s] := 1;
			END_IF;

			safeZone.DoorLock := lockDoor[n];
			safeZone.LiftGates := (safeZone.Zone_Status AND (safeZone.BagsInTransit OR NOT safeZone.AccessRequested)); // Edge protection gates.
			safeZone.HaltSys := NOT(safeZone.Zone_Status AND NOT safeZone.Disable);
		END_IF;

	END_FOR;

	IF NOT resetRequired[s] THEN
		masterResetRequest[s] := 0;
	END_IF;
	resetRequired[s] := 0;

	//Flash reset btn on main cabinet
	IF masterResetRequest[s] THEN // We can do a master reset and not out safe 0 to reset
		SafetyZone[startZone[s]].Main_Lamp := Std.Clock200ms;
	ELSE
		SafetyZone[startZone[s]].Main_Lamp := Std.Clock1s AND NOT SafetyZone[startZone[s]].Zone_Status;
	END_IF;

END_FOR;

END_PROGRAM
```

#### Variables.var - Local variables
```iecst
VAR CONSTANT
	MAX_SAFE_SYSTEMS : USINT := 2; (*Number of independant safety systems*)
END_VAR
VAR
	n : UINT;
	transitSettlePT : UDINT; (*Determines the amount of time to wait for bags in transit to settle before opening the interlock*)
	ton_10ms_Transit_Settle : ARRAY[0..MAX_SAFE_ZONES] OF TON_10ms; (*Determines the amount of time to wait for bags in transit to settle before opening the interlock*)
	safeState : ARRAY[0..MAX_SAFE_ZONES] OF USINT; (*USINT that tracks the state of the safe system so it can control the tower light*)
	debounceMasterPT : UDINT;
	masterReset : ARRAY[0..MAX_SAFE_ZONES] OF BOOL;
	ton_10ms_Master_Reset : ARRAY[0..MAX_SAFE_SYSTEMS] OF TON_10ms;
	masterResetRequest : ARRAY[0..MAX_SAFE_SYSTEMS] OF BOOL;
	startUpWarningPT : UDINT;
	ton_10ms_startUp_Warning : ARRAY[0..MAX_SAFE_SYSTEMS] OF TON_10ms;
	tp_10ms_reset_Pulse : TP_10ms;
	enableMasterReset : ARRAY[0..MAX_SAFE_SYSTEMS] OF BOOL;
	ton_10ms_Reset_Debounce : ARRAY[0..MAX_SAFE_ZONES] OF TON_10ms;
	ton_10ms_bagsInTransit : ARRAY[0..MAX_SAFE_ZONES] OF TON_10ms;
	f_trigRequestAccess : ARRAY[0..MAX_SAFE_ZONES] OF F_TRIG;
	ton_entryError : ARRAY[0..MAX_SAFE_ZONES] OF TON_10ms;
	resetRequired : ARRAY[0..MAX_SAFE_SYSTEMS] OF BOOL;
	lockDoor : ARRAY[0..MAX_SAFE_ZONES] OF BOOL;
	tof_HoistsOutOfPosition : ARRAY[0..MAX_SAFE_ZONES] OF TOF_10ms;
	safeZone : REFERENCE TO SafeZoneType;
	startZone : ARRAY[0..MAX_SAFE_SYSTEMS] OF UINT;
	endZone : ARRAY[0..MAX_SAFE_SYSTEMS] OF UINT;
	s : USINT;
	masterZone : BOOL;
	alarmCondition : ARRAY[0..MAX_SAFE_SYSTEMS] OF BOOL;
	tmrAlmOutput : ARRAY[0..MAX_SAFE_SYSTEMS] OF TON;
	masterZoneNo : UINT;
END_VAR
```

#### _decodeData.st
```iecst
ACTION _decodeData:

//	Zone Status Encoding
//	0 - Zone Input State
//	1 - Zone Ready FOR Reset
//	2 - E-stop FUB error
//	3 - EDM Input State
//	4 - EDM Ready
//	5 - EDM Error
//	6 - EDM Disabled
//	7 - Zone Dependancy
//	8 - Safe System OK
//	9 - Auto Reset
//	10 - ACCESS Request
//	11 - Zone Status

safeZone.Zone_Status 		:= safeZone.DataFromSafePLC.11;
safeZone.ResetReady			:= safeZone.DataFromSafePLC.1;
safeZone.RequestAccess		:= safeZone.DataFromSafePLC.10;   // Derived in the PLC from from Zone Healthy and Reset Push button

END_ACTION
```

### Passwords.txt
```
Development 	: safeplc
Commissioning 	: 123456
```

### mappSafety.var
```iecst
VAR
	MappSafety : MappSafety_typ;
END_VAR
```

### mappSafety.typ
```iecst
TYPE
	MappSafety_typ : 	STRUCT
		State : USINT;
		Commands : MappSafetyCommands_typ;
		Visu : MappSafetyVisu_typ;
	END_STRUCT;
	MappSafetyCommands_typ : 	STRUCT
		Transfer : BOOL;
		Complete : BOOL;
		Exchange : BOOL;
		Format : BOOL;
		Restart : BOOL;
		ActivateSetupMode : BOOL;
		ResetError : BOOL;
	END_STRUCT;
	MappSafetyVisu_typ : 	STRUCT
		Transfer : btn_ctrl_typ;
		Complete : btn_ctrl_typ;
		Exchange : btn_ctrl_typ;
		Format : btn_ctrl_typ;
		Restart : btn_ctrl_typ;
		ActivateSetupMode : btn_ctrl_typ;
		ResetError : btn_ctrl_typ;
	END_STRUCT;
	btn_ctrl_typ : 	STRUCT
		Enable : BOOL;
		Visible : BOOL;
	END_STRUCT;
END_TYPE
```

### Program Logical/Safety/mappSafety (IEC, version 1.00.1)

#### Main.st - Init, cyclic, exit code
```iecst
PROGRAM _INIT
	sfDomain := ADR(gSafeDomain);

	sfDomainConnect.UserName := 'Safety';
	sfDomainConnect.Password := 'safeplc';

	sfDomainTransfer.SafeAppFilePath :=	'SafeLOGIC-1'; // We must be connected for this to work.

	sfDomainConnect.SfDomain := sfDomainInfo.SfDomain := sfDomainTransfer.SfDomain := sfDomainControl.SfDomain :=  sfDomainExchange.SfDomain := sfDomainCompletion.SfDomain :=  sfDomain;
	refreshTime := T#5s;
	state ACCESS ADR(MappSafety.State);
	safeInfoValid := FALSE;
	state := 0;
END_PROGRAM

PROGRAM _CYCLIC

	sfDomainConnect.Enable := (state <> 200);
	IF NOT sfDomainConnect.Active AND (state <> 200) THEN  // No connection to the domain,
		safeInfoValid := 0;
	END_IF;

	sfDomainInfo.Execute 				:= 0;
	sfDomainTransfer.Execute 			:= 0;
	sfDomainCompletion.Execute 			:= 0;
	sfDomainExchange.Execute 			:= 0;
	sfDomainControl.Execute 			:= 0;

	ton_refresh(IN := (state = 10), PT:= refreshTime);

	CASE state OF
		0: // Connect to the safe PLC
			IF sfDomainConnect.Active THEN
				state := 1;
			ELSIF sfDomainConnect.Error THEN
				state := 200;
			END_IF;

		1: // Read the status of the safety plc.
			sfDomainInfo.Execute := 1;
			IF sfDomainInfo.Done THEN
				safeInfoValid := 1;
				safetyInfo := sfDomainInfo.Info;
				state := 10;
			ELSIF sfDomainInfo.Error THEN
				state := 200;
			END_IF;

		10:// Decide what to do//
			// Check for any actions first.
			IF NOT  safetyInfo.SafeApplication.ExistOnSafeLogic THEN
				state := 11;
			ELSIF MappSafety.Commands.Transfer THEN
				MappSafety.Commands.Transfer := 0;
				state := 20;
			ELSIF MappSafety.Commands.Complete THEN
					MappSafety.Commands.Complete := 0;
					state := 30;
			ELSIF MappSafety.Commands.Exchange THEN
				MappSafety.Commands.Exchange := 0;
				state := 40;
			ELSIF MappSafety.Commands.Restart THEN
				MappSafety.Commands.Restart := 0;
				state := 50;
			ELSIF MappSafety.Commands.Format THEN
				MappSafety.Commands.Format := 0;
				state := 51;
			ELSIF MappSafety.Commands.ActivateSetupMode THEN
				MappSafety.Commands.ActivateSetupMode := 0;
				state := 52;
			ELSIF ton_refresh.Q THEN
				state := 1;
			END_IF;

		11:// Program not downloaded.
			IF MappSafety.Commands.Transfer THEN
				MappSafety.Commands.Transfer := 0;
				state := 20;
			ELSIF MappSafety.Commands.Restart THEN
				MappSafety.Commands.Restart := 0;
				state := 50;
			ELSIF MappSafety.Commands.Format THEN
				MappSafety.Commands.Format := 0;
				state := 51;
			END_IF;

		20:// Transfer the project.
			sfDomainTransfer.Execute := 1;
			IF sfDomainTransfer.Done THEN
				state := 0;
			ELSIF sfDomainTransfer.Error THEN
				state := 200;
			END_IF;

		30:// Complete the setup
			sfDomainCompletion.Execute := 1;
			IF sfDomainCompletion.Done THEN
				state := 0;
			ELSIF sfDomainCompletion.Error THEN
				state := 200;
			END_IF;

		40:// Acknowledge some request from the safe PLC.
			sfDomainExchange.Execute := 1;
			IF sfDomainExchange.Done THEN
				state := 0;
			ELSIF sfDomainExchange.Error THEN
				state := 200;
			END_IF;

		50:// Control the Safe PLC -- Force a restart..
			sfDomainControl.Execute := 1;
			sfDomainControl.ControlCommand := sfDOM_REBOOT;
			IF sfDomainControl.Done THEN
				state := 0;
			ELSIF sfDomainControl.Error THEN
				state := 200;
			END_IF;

		51:// Control the Safe PLC -- Format the safe plc
			sfDomainControl.Execute := 1;
			sfDomainControl.ControlCommand := sfDOM_FORMAT_REBOOT;
			IF sfDomainControl.Done THEN
				state := 0;
			ELSIF sfDomainControl.Error THEN
				state := 200;
			END_IF;

		52:// Control the Safe PLC -- Activate setup mode.
			sfDomainControl.Execute := 1;
			sfDomainControl.ControlCommand := sfDOM_ACT_SETUP_MODE;
			IF sfDomainControl.Done THEN
				state := 0;
			ELSIF sfDomainControl.Error THEN
				state := 200;
			END_IF;

		200:// Error step
			IF MappSafety.Commands.ResetError THEN
				MappSafety.Commands.ResetError := 0;
				state := 0;
			END_IF;
	END_CASE;

	sfDomainCompletion.Info := safetyInfo;
	sfDomainExchange.Info := safetyInfo;

	sfDomainConnect();
	sfDomainInfo();
	sfDomainTransfer();
	sfDomainControl();
	sfDomainExchange();
	sfDomainCompletion();

	//We have to read the domain info and pass it to the Completion function.
	_visu;

END_PROGRAM
PROGRAM _EXIT

	sfDomainConnect.Enable 					:= 0;
	sfDomainConnect();

END_PROGRAM
```

#### _visu.st
```iecst
ACTION _visu:

	brsitoa(MappSafety.State,ADR(sState));
	brsitoa(safetyInfo.Status.SafeOSState,ADR(sSafeOsState));
	brsitoa(safetyInfo.Status.SafeNodesState,ADR(sSafeNodeState));
	brsitoa(safetyInfo.Status.SystemState,ADR(sSystemState));
	brsitoa(safetyInfo.Status.OperationalModeState,ADR(sOperationalModeState));

	MappSafety.Visu.ResetError.Enable := MappSafety.Visu.ResetError.Visible	:=  (MappSafety.State = 200);

	MappSafety.Visu.Transfer.Enable 			:= NOT MappSafety.Commands.Transfer AND (MappSafety.State <= 11);
	MappSafety.Visu.Complete.Enable 			:= NOT MappSafety.Commands.Complete AND (MappSafety.State <= 10);
	MappSafety.Visu.ActivateSetupMode.Enable 	:= NOT MappSafety.Commands.ActivateSetupMode AND (MappSafety.State <= 10);
	MappSafety.Visu.Exchange.Enable 			:= NOT MappSafety.Commands.Exchange AND (MappSafety.State <= 10);
	MappSafety.Visu.Format.Enable 				:= NOT MappSafety.Commands.Format AND (MappSafety.State <= 11);
	MappSafety.Visu.Restart.Enable 				:= NOT MappSafety.Commands.Restart AND (MappSafety.State <= 10);

	MappSafety.Visu.Exchange.Visible 	:= MappSafety.Visu.ActivateSetupMode.Visible := safeInfoValid AND NOT safetyInfo.Status.SetupModeActive AND (MappSafety.State <= 10);
	MappSafety.Visu.Transfer.Visible 	:= safeInfoValid;// AND safetyInfo.SafeApplication.ExistOnSafeLogic;
	MappSafety.Visu.Complete.Visible 	:= safeInfoValid AND (safetyInfo.SafeApplication.ExistOnSafeLogic AND NOT safetyInfo.SafeApplication.Acknowledged) OR safetyInfo.Status.SetupModeActive ;
	MappSafety.Visu.Restart.Visible 	:= 	TRUE;
	MappSafety.Visu.Format.Visible 		:= safeInfoValid;// AND safetyInfo.SafeApplication.ExistOnSafeLogic;

END_ACTION
```

#### Variables.var - Local variables
```iecst
VAR
	sfDomain : UDINT;
	sfDomainInfo : SfDomainInfo;
	sfDomainTransfer : SfDomainTransfer;
	sfDomainCompletion : SfDomainCompletion;
	sfDomainControl : SfDomainControl;
	sfDomainExchange : SfDomainExchange;
	sfDomainConnect : SfDomainConnect;
	safetyInfo : SfDomainInfoType;
	refreshTime : TIME;
	ton_refresh : TON;
	state : REFERENCE TO USINT;
	sState : STRING[5];
	sSafeOsState : STRING[5];
	sSafeNodeState : STRING[5];
	sSystemState : STRING[5];
	sOperationalModeState : STRING[5];
	safeInfoValid : BOOL;
END_VAR
```

### Inwatec.var
```iecst
VAR CONSTANT
	INWATEC_RELEASE_TO : USINT := 0; (*DROP INTO INWATEC*)
	INWATEC_RECIEVE_FROM : USINT := 1; (*RECIEVE FROM INWATEC*)
END_VAR
VAR
	Inwatec : ARRAY[0..MAX_INWATEC_INTERFACES] OF Inwatec_typ;
END_VAR
VAR CONSTANT
	MAX_INWATEC_INTERFACES : UINT := 11;
END_VAR
```

### Inwatec_Interface.typ
```iecst
TYPE
	Inwatec_typ : 	STRUCT
		Inlet : Inwatec_data_typ;
		Outlet : Inwatec_data_typ;
		Config : Inwatec_config_typ;
	END_STRUCT;
	Inwatec_config_typ : 	STRUCT
		ServerURL : STRING[255];
		Direction : USINT; (*0 = drop to inwatec, 1= recieve from inwatec*)
		Authenication : UAUserIdentityToken := (UserIdentityTokenType:=UAUITT_Username,TokenParam1:='ExternalSystem',TokenParam2:='Inwatec');
		CommID : USINT;
	END_STRUCT;
	Inwatec_data_typ : 	STRUCT
		tx_handshake : USINT;
		option_flag_1 : USINT;
		option_flag_2 : USINT;
		system_status : USINT;
		i_am_alive : BOOL;
		batch_id : UDINT;
		source_id : DINT;
		batch_count : INT;
		weight : REAL;
		customer : STRING[25];
		customer_name : STRING[25];
		customer_numeric : DINT;
		category : STRING[20];
		category_name : STRING[20];
		category_numeric : DINT;
		lot : STRING[20];
		lot_numeric : DINT;
		sublot : STRING[20];
		sublot_numeric : DINT;
		option_1 : UDINT;
		option_2 : DINT;
	END_STRUCT;
END_TYPE
```

### Variables.var
```iecst
VAR
	OPCuA_Client : ARRAY[0..MAX_OPCuA_CLIENTS] OF OPCuaClient_typ;
END_VAR
```

### Types.typ
```iecst
TYPE
	OPCuaClient_typ : 	STRUCT
		State : UINT;
		Config : OPCuAClient_Config_typ;
		Functions : OPCuaClient_Functions_typ;
		Error : OPCuaClient_Error_typ;
		WriteData : OPCuAClient_WriteData_typ;
		ReadData : OPCuAClient_ReadData_typ;
	END_STRUCT;
	OPCuAClient_Config_typ : 	STRUCT
		ServerURL : STRING[255];
		SessionInfo : UASessionConnectInfo;
		SessionUser : UAUserIdentityToken;
		Data : OPCuAClient_Confg_Data_typ;
	END_STRUCT;
	OPCuAClient_WriteData_typ : 	STRUCT
		NodeID : ARRAY[0..MAX_WRITE_NODES]OF UANodeID;
		NodeInfo : ARRAY[0..MAX_WRITE_NODES]OF UANodeAdditionalInfo;
		Variable : ARRAY[0..MAX_WRITE_NODES]OF STRING[MAX_LENGTH_VARIABLE];
		ErrorID : ARRAY[0..MAX_WRITE_NODES]OF DWORD;
		TimeStamps : ARRAY[0..MAX_WRITE_NODES]OF DATE_AND_TIME;
	END_STRUCT;
	OPCuAClient_ReadData_typ : 	STRUCT
		NodeID : ARRAY[0..MAX_READ_NODES]OF UANodeID;
		NodeInfo : ARRAY[0..MAX_READ_NODES]OF UANodeAdditionalInfo;
		Variable : ARRAY[0..MAX_READ_NODES]OF STRING[MAX_LENGTH_VARIABLE];
		ErrorID : ARRAY[0..MAX_READ_NODES]OF DWORD;
		TimeStamps : ARRAY[0..MAX_READ_NODES]OF DATE_AND_TIME;
	END_STRUCT;
	OPCuaClient_Functions_typ : 	STRUCT
		Connect : UA_Connect;
		GetNameSpace : UA_GetNamespaceIndex;
		WriteBulk : UaClt_WriteBulk;
		ReadBulk : UaClt_ReadBulk;
		Disconnect : UA_Disconnect;
		RetryTimer : TON;
		ErrorStatePLS : R_TRIG;
	END_STRUCT;
	OPCuaClient_Error_typ : 	STRUCT
		ErrorID : DWORD; (**Raw error info*)
		ErrorCode : UINT; (**Decoded Error message*)
		Message : STRING[254];
		ErrorState : UINT; (*State which caused the error*)
		ErrorNode : UINT; (*Index of the read or write node that caused the error*)
	END_STRUCT;
	OPCuAClient_Confg_Data_typ : 	STRUCT
		Read : ARRAY[0..MAX_READ_NODES]OF OPCuAClient_Config_ReadData_typ;
		Write : ARRAY[0..MAX_WRITE_NODES]OF OPCuAClient_Confg_WriteData_typ;
		WriteCount : UINT;
		ReadCount : UINT;
	END_STRUCT;
	OPCuAClient_Confg_WriteData_typ : 	STRUCT
		NodeID : UANodeID;
		NodeInfo : UANodeAdditionalInfo;
		Variable : STRING[MAX_LENGTH_VARIABLE];
		ErrorID : DWORD;
		TimeStamps : DATE_AND_TIME;
	END_STRUCT;
	OPCuAClient_Config_ReadData_typ : 	STRUCT
		NodeID : UANodeID;
		NodeInfo : UANodeAdditionalInfo;
		Variable : STRING[MAX_LENGTH_VARIABLE];
		ErrorID : DWORD;
		TimeStamps : DATE_AND_TIME;
	END_STRUCT;
END_TYPE
```

### Constants.var
```iecst
(*STATES*)
VAR CONSTANT
	OPCuA_CLIENT_STATE_CONNECT : UINT := 0;
	OPCuA_CLIENT_STATE_GET_NAMESPACE : UINT := 1;
	OPCuA_CLIENT_STATE_BUILD_DATA : UINT := 2;
	OPCuA_CLIENT_STATE_READ_WRITE : UINT := 3;
	OPCuA_CLIENT_STATE_DISCONNECT : UINT := 4;
	OPCuA_CLIENT_STATE_ERROR : UINT := 16#FFFF;
END_VAR
(*CONFIG*)
VAR CONSTANT
	MAX_WRITE_NODES : UINT := 20;
	MAX_READ_NODES : UINT := 20;
	MAX_OPCuA_CLIENTS : UINT := 11;
END_VAR
```

### ErrorConstants.var
```iecst
VAR CONSTANT
	OPCuA_ERR_OUT_OF_SERVICE : DWORD := 16#80AD0000;
	OPCuA_ERR_INVALID_HDL : DWORD := 16#A0080000;
	OPCuA_ERR_BAD_CONNECTION : DWORD := 16#80050000;
	OPCuA_ERR_TIMEOUT : DWORD := 16#800A0000;
END_VAR
```
